	WorkAreaState^[WorkAreaNumber].Supporto := Forming^[1].Pallet;
	WorkAreaState^[WorkAreaNumber].F := 1;
	WorkAreaState^[WorkAreaNumber].ID 	:= ProgressiveNrWA^;
	ProgressiveNrWA^ := ProgressiveNrWA^ + 1;
	WorkAreaState^[WorkAreaNumber].P 	:= 0;
	WorkAreaState^[WorkAreaNumber].Slow := 1;
	WorkAreaState^[WorkAreaNumber].LGVAttr := Forming^[WorkAreaState^[WorkAreaNumber].F].LGVAttr;
	WorkAreaState^[WorkAreaNumber].State := WORKAREA_STATE_OCCUPIED_WORKING;
	
	InserisciNuovoPallet := FALSE;

ELSIF InserisciNuovoPallet AND WorkAreaState^[WorkAreaNumber].State < WORKAREA_STATE_OCCUPIED_WORKING AND FALSE THEN
	
	//Se la postazione ha codice fisso, lo assegno!
	IF CodicePostazione = 0 AND WorkAreaCodiciFissi[WorkAreaNumber] > 0 THEN
		CodicePostazione := WorkAreaCodiciFissi[WorkAreaNumber];
	END_IF

	(* Cerco Formatura *)
	IndiceFormaturaPostazione := 0;
	IndiceFormaturaPostazione := TFPalletizerGetFormingFromCodeSlab(Forming,CodicePostazione);
	//Assegno la formatura successivamanete nel WAManager
	IF IndiceFormaturaPostazione < 1 THEN
		IndiceFormaturaPostazione := 0;
		//Valuto la zona della postazione e ricavo la formatura in base alla zona di appartenenza	
	
		FOR cod:=1 TO MAXFORMINGCODE DO
			FormaturaZona[cod] := 0;
		END_FOR
		DoppiaFormaturaAttiva := FALSE;
		CodiceInFormaturaMem := 0;
		NumCodiciInFormaturaAttiviPerZona := 0;
		FOR zone:=1 TO MAXZONE DO
			FOR ar:=1 TO MAXAREA DO
				(* Verifico se la WorkArea appartiena ad una Zona *)
				IF WorkAreaZone.Zone[zone].WorkArea[ar] = WorkAreaNumber THEN
					FOR cod:=1 TO MAXFORMINGCODE DO
						IF FormaturaZona[cod] > 0 THEN
							DoppiaFormaturaAttiva := TRUE;
						END_IF
						FormaturaZona[cod] := TFPalletizerGetFormingFromCodeSlab(Forming,WorkAreaZone.Zone[zone].Code[cod]);
						IF WorkAreaZone.Zone[zone].Code[cod] <> CodiceInFormaturaMem  THEN//Memorizzo se ho un codice 
							NumCodiciInFormaturaAttiviPerZona := NumCodiciInFormaturaAttiviPerZona+1;
							CodiceInFormaturaMem := WorkAreaZone.Zone[zone].Code[cod];
						END_IF
					END_FOR
					EXIT;//Esco e vado a valutare le formature
				END_IF
			END_FOR
		END_FOR	
		FOR ar:=1 TO 4 DO
			FormaturePresenti[ar] := 0;
		END_FOR
		FOR ar:=1 TO MAXFORMINGCODE DO
		
			CASE FormaturaZona[ar] OF
				1:
					FormaturePresenti[1] := FormaturePresenti[1]+1; 	
				2:
					FormaturePresenti[2] := FormaturePresenti[2]+1;
				3:
					FormaturePresenti[3] := FormaturePresenti[3]+1;
				4:
					FormaturePresenti[4] := FormaturePresenti[4] +1;
			ELSE
				IndiceFormaturaPostazione := 0;			
			END_CASE				
		END_FOR
		//Cerco se nella zona ci sono + formature presenti, se è così codice formatura = 0, in modo che la macchina lo assagne in base alle esigenze
		//Altrimenti se solo una formatura è presente gli assegno quella!			
		IF FormaturePresenti[1] >= 1 THEN
			IF FormaturePresenti[2] >= 1 OR FormaturePresenti[3] >= 1 OR FormaturePresenti[4] >= 1 OR DoppiaFormaturaAttiva THEN
				IndiceFormaturaPostazione := 0;
			ELSE
				IndiceFormaturaPostazione := 1;
				IF NumCodiciInFormaturaAttiviPerZona = 1 THEN
					 CodicePostazione := CodiceInFormaturaMem;
				END_IF
			END_IF		
		ELSIF FormaturePresenti[2] >= 1 THEN
			IF FormaturePresenti[1] >= 1 OR FormaturePresenti[3] >= 1 OR FormaturePresenti[4] >= 1 OR DoppiaFormaturaAttiva THEN
				IndiceFormaturaPostazione := 0;
			ELSE
				IndiceFormaturaPostazione := 2;
				IF NumCodiciInFormaturaAttiviPerZona = 1 THEN
					 CodicePostazione := CodiceInFormaturaMem;
				END_IF
			END_IF		
		ELSIF FormaturePresenti[3] >= 1 THEN
			IF FormaturePresenti[2] >= 1 OR FormaturePresenti[1] >= 1 OR FormaturePresenti[4] >= 1 OR DoppiaFormaturaAttiva THEN
				IndiceFormaturaPostazione := 0;
			ELSE
				IndiceFormaturaPostazione := 3;
				IF NumCodiciInFormaturaAttiviPerZona = 1 THEN
					 CodicePostazione := CodiceInFormaturaMem;
				END_IF
			END_IF		
		ELSIF FormaturePresenti[4] >= 1 THEN
			IF FormaturePresenti[2] >= 1 OR FormaturePresenti[3] >= 1 OR FormaturePresenti[1] >= 1 OR DoppiaFormaturaAttiva THEN
				IndiceFormaturaPostazione := 0;
			ELSE
				IndiceFormaturaPostazione := 4;
				IF NumCodiciInFormaturaAttiviPerZona = 1 THEN
					 CodicePostazione := CodiceInFormaturaMem;
				END_IF
			END_IF		
		END_IF
	END_IF
	
	WorkAreaState^[WorkAreaNumber].Taped := -1;
	WorkAreaState^[WorkAreaNumber].LGV_ReqAbort := FALSE;
	IF AbilitaAssegnazioneCodicePiazzoleConPaccoSuRibaltino AND CodicePostazione = 0 THEN
		WorkAreaState^[WorkAreaNumber].Code := 0;
		WorkAreaState^[WorkAreaNumber].Initialize := TRUE;
	ELSE
		WorkAreaState^[WorkAreaNumber].Code := CodicePostazione;
		WorkAreaState^[WorkAreaNumber].Initialize := FALSE;
	END_IF
	WorkAreaState^[WorkAreaNumber].Supporto := Forming^[IndiceFormaturaPostazione].Pallet;
	WorkAreaState^[WorkAreaNumber].F := IndiceFormaturaPostazione;
	
	WorkAreaState^[WorkAreaNumber].ID := ProgressiveNrWA^;
	ProgressiveNrWA^ := ProgressiveNrWA^ + 1;
	WorkAreaState^[WorkAreaNumber].P := 0;
	WorkAreaState^[WorkAreaNumber].Slow := 1;
	WorkAreaState^[WorkAreaNumber].LGVAttr := Forming^[WorkAreaState^[WorkAreaNumber].F].LGVAttr;
	WorkAreaState^[WorkAreaNumber].State := WORKAREA_STATE_OCCUPIED_WORKING;

	InserisciNuovoPallet := FALSE;
END_IF

END_FUNCTION_BLOCK

// ---- POUs/TFPalletizerData/TFClearWorkAreaArray.TcPOU
FUNCTION TFClearWorkAreaArray : BOOL
VAR_INPUT
	WorkArea : POINTER TO ARRAY [1..MAXAREA] OF TFMachinePalletizer_WorkArea;
	WorkAreaState : POINTER TO ARRAY [1..MAXAREA] OF TFMachinePalletizer_WorkAreaState;
	k : uINT;
END_VAR
VAR
END_VAR

(* Copia dello stato delle WA in un backup *)
IF WorkAreaState^[k].ID > 0 THEN
	WorkAreaStateBK[k] := WorkAreaState^[k];
END_IF

WorkAreaState^[k] := EmptyWorkAreaState;
WorkAreaState^[k].State		:= WORKAREA_STATE_FREE_ENABLED;	(* Stato Area di Lavoro/Piazzola
																			(0=Assente e Area Disabilitata,
																			1=Presente e Area Disabilitata,
																			2=Assente in Lavorazione,
																			3=Presente in Lavorazione,
																			4=Presente con Pallettizzazione Terminata,
																			5=Presente con Pallettizzazione Terminata e Area Disabilitata,
																			6=Presente in Nastratura,
																			7=Presente in Nastratura e Area Disabilitata,
																			8=Presente con Nastratura Terminata,
																			9=Presente con Nastratura Terminata e Area Disabilitata,
																			10=Presente con Lavorazione Terminata,
																			11=Presente con Lavorazione Terminata e Area Disabilitata,
																			12=Presente con LGV in Richiesta Ingresso,
																			13=Presente con LGV in Richiesta Ingresso e Area Disabilitata,
																			14=Presente con LGV in Ingombro,
																			15=Presente con LGV in Ingombro e Area Disabilitata,
																			16=Presente con LGV Fuori Ingombro e Pallet Estratto,
																			17=Presente con LGV Fuori Ingombro e Pallet Estratto e Area Disabilitata, NOT USED !!!!!!!!!!!
																			99=Errore
																			-1 dato non valido) *)
																			
//TFClearWorkAreaStateSlab(WorkAreaState,k);																			
																			
WorkAreaState^[k].F					:= -1;	(* Forming Pointer - Puntatore tabella formature (1..n=, -1 dato non valido *)
WorkAreaState^[k].P					:= -1;	(* Pack Pointer - Puntatore tabella ELEMENTO (0..n-1=, -1 dato non valido),Numero ELEMENTO successivo da depositare *)
              
WorkAreaState^[k].Code				:= -1;	(* Codice di Pallettizzazione (0..n=, -1 dato non valido) x lastre, se Magazzino Falde, codice della falda *)
              
WorkAreaState^[k].PackPointerModified	:= FALSE;		(* Se TRUE, indica che è stata effettuata una modfica sui dati della WA da parte dell' HMI (Settata da HMI e resettata da PLC) *)
WorkAreaState^[k].PackPointer			:= -1;			(* Rappresenta l'indice del pacco da depositare dopo modfica manuale,cioè con PackPointerModified=TRUE *)

WorkAreaState^[k].Slab := EmptySlabArray;

WorkAreaState^[k].LGVAttr				:= 0;

TFClearWorkAreaBCRead(WorkAreaState);//Resetto i vari stati dl BARCODE

WorkAreaState^[k].H					:= 0.0; (* (mm) Altezza Reale. Viene calcolata dal PLC dopo ogni prelievo (Vuoti o Falde) o deposito Pallet e durante la pallettizzazione *)
WorkAreaState^[k].HPL				:= 0.0; (* (mm) Altezza del pallett utilizzato + altezza layers utilizzati *)

TFClearApprendimento(ADR(WorkAreaState^[k].Apprendimento));//Azzeramento apprendimento

(*
(* Apprendimenti nelle varie direzioni *)
WorkAreaState^[k].DoLearn_Y0		:= APPRENDIMENTO_DA_ESEGUIRE;	(* Stato apprendimento Direzione Y LATO 0° 0=Disabilitato, 1=Abilitato da Eseguire, 2=Eseguito, -1 dato non valido *)
WorkAreaState^[k].Learn_Y0			:= 0.0;	(* (mm) Quota inizio Apprendimento Direzione Y LATO 0° *)
WorkAreaState^[k].Learned_Y0		:= 0.0; (* Quota rilevata durante apprendimento Direzione Y LATO 0° *)

WorkAreaState^[k].DoLearn_Y180		:= APPRENDIMENTO_DA_ESEGUIRE;	(* Stato apprendimento Direzione Y LATO 180° 0=Disabilitato, 1=Abilitato da Eseguire, 2=Eseguito, -1 dato non valido *)
WorkAreaState^[k].Learn_Y180		:= 0.0;	(* (mm) Quota inizio Apprendimento Direzione Y LATO 180° *)
WorkAreaState^[k].Learned_Y180		:= 0.0; (* Quota rilevata durante apprendimento Direzione Y LATO 180° *)

WorkAreaState^[k].DoLearn_Z			:= APPRENDIMENTO_DA_ESEGUIRE;	(* Stato apprendimento Direzione Z 0=Disabilitato, 1=Abilitato da Eseguire, 2=Eseguito, -1 dato non valido *)
WorkAreaState^[k].Learn_Z			:= 0.0;	(* (mm) Quota inizio Apprendimento Direzione Z *)
WorkAreaState^[k].Learned_Z			:= 0.0; (* Quota rilevata durante apprendimento Direzione Z *)
*)
WorkAreaState^[k].RefuseLGV       	:= FALSE;	(* Abilitazione chiamata LGV a termine pallettizzazione - TRUE= Non chiama LGV quando pallet pieno, FALSE= viene eseguita richiesta LGV *)
              
WorkAreaState^[k].LGV_Req			:= 0;	(* Richiesta LGV (0=Nop, 1=Richiesta LGV, 2= Consenso Ingresso, -1= non valido) *)
WorkAreaState^[k].LGV_GetIn_GetOut	:= 0;	(* Tipo Richiesta LGV  (0=Nop, 1=Richiesta Prelievo, 2= Richiesta Deposito, -1= non valido) *)	
WorkAreaState^[k].LGV_ReqAbort		:= FALSE; (* Aborto chimata LGV *)


TFClearWorkAreaArray := TRUE;

END_FUNCTION

// ---- POUs/TFPalletizerData_Lastre/TFClearWorkAreaBCRead.TcPOU
FUNCTION TFClearWorkAreaBCRead : BOOL
VAR_INPUT
	WorkAreaState : POINTER TO TFMachinePalletizer_WorkAreaState;
END_VAR
VAR
	i : INT;
END_VAR

FOR i:=1 TO MAXNUMBARCODE DO
	WorkAreaState^.BCRead[i].State := LETTURA_ESEGUITA;
	WorkAreaState^.BCRead[i].Value := ''; 
	WorkAreaState^.BCRead[i].ErrorCode := 0;
END_FOR
TFClearWorkAreaBCRead := TRUE;

END_FUNCTION

// ---- POUs/TFPalletizerData_Lastre/TFClearApprendimento.TcPOU
FUNCTION TFClearApprendimento : BOOL //Funzione che pulisce la struttura dell'apprendimento
VAR_INPUT
	Apprendimento : POINTER TO TFMachinePalletizer_CoordinateApprendimento;
END_VAR
VAR
	i : INT;
END_VAR

MEMSET(ADR(Apprendimento^),0,SIZEOF(Apprendimento^));
TFClearApprendimento := TRUE;

END_FUNCTION

// ---- POUs/TFPalletizerData_Lastre/TFPalletizerGetFormingFromCodeSlab.TcPOU
FUNCTION TFPalletizerGetFormingFromCodeSlab : INT
VAR_INPUT
	Forming : POINTER TO ARRAY [1..MAXFORMING] OF TFMachinePalletizer_FormingForSlab;
	FCode : INT;
END_VAR
VAR
	pp : UINT;
	pf : INT;
	PCode : UINT;
END_VAR

(* Per Tutte le Formature Attive *)
FOR pf:=1 TO MAXFORMING DO
	IF Forming^[pf].Enable = 1 THEN
		(* Per tutti i codici di Pallettizzazione *)
		FOR pp:=1 TO MAXFORMINGCODE DO
			IF Forming^[pf].Code[pp] = FCode THEN
				TFPalletizerGetFormingFromCodeSlab := pf;
				RETURN;
			END_IF
		END_FOR
	END_IF
END_FOR
TFPalletizerGetFormingFromCodeSlab := 0;

END_FUNCTION

// ---- POUs/TFPalletizerDataTF/Utility Varie/TFCalcolaNumeroPostazioneDXSX.TcPOU
FUNCTION_BLOCK TFCalcolaNumeroPostazioneDXSX (* Restituisce il numero della postazione a DX e a SX rispetto alla poszione attuale della pinza *)
VAR_INPUT
	WorkArea 					: POINTER TO ARRAY[1..MAXAREA] OF TFMachinePalletizer_WorkArea; //Puntatore alla struttura WorkArea
	PosizioneAttuale			: LREAL;	//Posizione attuale dell'asse X
	DirezioneAsseX_Positiva		: BOOL;
END_VAR
VAR_OUTPUT
	NPostazioneDX : UINT;
	NPostazioneSX : UINT;
	PostazionePartenza : UINT;
END_VAR
VAR
	WADX: UINT;
	WASX: UINT;
	waDXSX : UINT;
END_VAR
(* Restituisce il numero della postazione a DX e a SX rispetto alla poszione attuale della pinza *)

WASX := 0;
WADX := 0;

CASE VERSO_PALLETTIZZATORE OF
	PALLETTIZZATORE_DX :
						FOR waDXSX := 1 TO MAXAREAPRESENT DO
							IF PosizioneAttuale > WorkArea^[waDXSX].X + 50  THEN
								WADX := WADX +1;
								IF WADX > MAXAREAPRESENT THEN
									WADX := MAXAREAPRESENT;
								END_IF
								NPostazioneDX		:= WADX;
								WorkAreaDX_Attuale  := WADX;
							ELSE
								WASX := WADX + 1;
								IF WADX = 0 THEN
									WADX:=1;
								END_IF
								IF WASX > MAXAREAPRESENT THEN
									WASX := MAXAREAPRESENT;
								END_IF
								NPostazioneSX		:= WASX;
								WorkAreaSX_Attuale := WASX;
								IF DirezioneAsseX_Positiva THEN
									PostazionePartenza:= WADX+1;
								ELSE
									PostazionePartenza:= WASX-1;
									
								END_IF
								EXIT;
							END_IF
						END_FOR					
						
	
	PALLETTIZZATORE_SX :
						CASE ORDINE_DISPOSIZIONE_POSTAZIONI OF

							CRESCENTE:
										FOR waDXSX := 1 TO MAXAREAPRESENT DO
											IF PosizioneAttuale > WorkArea^[waDXSX].X + 50  THEN
												WADX := WADX +1;
												IF WADX > MAXAREAPRESENT THEN
													WADX := MAXAREAPRESENT;
												END_IF
												NPostazioneDX		:= WADX;
												WorkAreaDX_Attuale  := WADX;
											ELSE
												WASX := WADX + 1;
												IF WADX = 0 THEN
													WADX:=1;
												END_IF
												IF WASX > MAXAREAPRESENT THEN
													WASX := MAXAREAPRESENT;
												END_IF
												NPostazioneSX		:= WASX;
												WorkAreaSX_Attuale := WASX;
												IF DirezioneAsseX_Positiva THEN
													
													//PostazionePartenza:= WADX;
													PostazionePartenza:= WASX;
												ELSE
													//PostazionePartenza:= WASX;
													PostazionePartenza:= WASX;
												END_IF
												EXIT;
											END_IF
										END_FOR
										
							DECRESCENTE:
										FOR waDXSX := MAXAREAPRESENT  TO 1 BY -1 DO
											IF PosizioneAttuale > WorkArea^[waDXSX].X THEN
												IF waDXSX = MAXAREAPRESENT THEN
													NPostazioneSX		:= 99;//Punto di prelievo
													WorkAreaSX_Attuale  := 99;
													NPostazioneDX		:= waDXSX;
													WorkAreaDX_Attuale  := waDXSX;
												ELSIF waDXSX = 1 THEN
													NPostazioneSX		:= 1;
													NPostazioneDX		:= 1;
													WorkAreaSX_Attuale  := 1;
													WorkAreaDX_Attuale  := 1;
													IF DirezioneAsseX_Positiva THEN
														PostazionePartenza:= WorkAreaDX_Attuale;
													ELSE
														PostazionePartenza:= WorkAreaSX_Attuale;
													END_IF
													EXIT;
												ELSE
													NPostazioneSX		:= waDXSX+1;
													NPostazioneDX		:= waDXSX-1;
													WorkAreaSX_Attuale  := waDXSX;
													WorkAreaDX_Attuale	:= waDXSX;
												END_IF	
												
											ELSIF PosizioneAttuale <= WorkArea^[waDXSX].X THEN
												IF waDXSX = MAXAREAPRESENT THEN
													NPostazioneSX		:= 99;//Punto di prelievo
													NPostazioneDX		:= waDXSX;
													WorkAreaSX_Attuale  := waDXSX;
													WorkAreaDX_Attuale  := waDXSX;
													IF DirezioneAsseX_Positiva THEN
														PostazionePartenza:= WorkAreaDX_Attuale;
													ELSE
														PostazionePartenza:= WorkAreaSX_Attuale;
													END_IF
													EXIT;
												ELSIF waDXSX = 1 THEN
													NPostazioneSX		:= waDXSX+1;
													NPostazioneDX		:= 1;
													WorkAreaSX_Attuale  := waDXSX;
													WorkAreaDX_Attuale  := waDXSX;
												ELSE
													NPostazioneSX		:= waDXSX+1;
													NPostazioneDX		:= waDXSX-1;
													WorkAreaSX_Attuale  := waDXSX;
													WorkAreaDX_Attuale	:= waDXSX;
													IF DirezioneAsseX_Positiva THEN
														PostazionePartenza:= WorkAreaDX_Attuale;
													ELSE
														PostazionePartenza:= WorkAreaSX_Attuale;
													END_IF
													EXIT;
												END_IF
												
											END_IF
										END_FOR	
										
						END_CASE
	
	
END_CASE

END_FUNCTION_BLOCK

// ---- Data types/AlbertoPruevas/Funciones/Fun_SensoresTasteggio.TcPOU
FUNCTION Fun_SensoresTasteggio : BOOL
VAR_INPUT
	Sensor_Tasteo_1 				: BOOL ;
	Sensor_Tasteo_2 				: BOOL ;
	Sensor_Tasteo_3 				: BOOL ;
	Sensor_Tasteo_4 				: BOOL ;
	Nu_sensores_Dar_Out				: BYTE ;
END_VAR
VAR_OUTPUT
	Sensores_Tasteggio_Ok 			: BOOL ;
	Nu_Sesores_Activos				: BYTE ;
END_VAR
VAR
END_VAR

Nu_Sesores_Activos := BOOL_TO_BYTE(Sensor_Tasteo_1) + BOOL_TO_BYTE(Sensor_Tasteo_2) + BOOL_TO_BYTE(Sensor_Tasteo_3) + BOOL_TO_BYTE(Sensor_Tasteo_4) ; 

IF Nu_Sesores_Activos >= Nu_sensores_Dar_Out THEN
	Sensores_Tasteggio_Ok := TRUE ;
	ELSE
	Sensores_Tasteggio_Ok := FALSE ;	
	
END_IF

END_FUNCTION

// ---- Data types/AlbertoPruevas/Funciones/Fun_PiezaLadoCaballete.TcPOU
FUNCTION Fun_PiezaLadoCaballete : Uint
VAR_INPUT
	Nu_PiezaGlobal 			: UINT ;
	Grados 					: pointer TO UINT ;
END_VAR
VAR_OUTPUT
	Nu_pieza_LadoA: UINT;
	Nu_pieza_LadoB: UINT;
END_VAR
VAR
	
	RestoDiv: UINT;
END_VAR



//Dia 23-10-2025
CASE Nu_PiezaGlobal OF
	1:
		Nu_pieza_LadoA :=  Nu_PiezaGlobal ;
		Grados^ := 0;
	2..100 :
		IF Nu_PiezaGlobal > 1 THEN 
			RestoDiv := Nu_PiezaGlobal MOD 2 ;
			CASE RestoDiv OF
				0:
					Nu_pieza_LadoB := Nu_PiezaGlobal / 2 ;
					Grados^ := 180;
				1:
					Nu_pieza_LadoA := ((Nu_PiezaGlobal-1) / 2)+1 ;
					Grados^ := 0;	
			END_CASE
		END_IF
END_CASE

END_FUNCTION

// ---- POUs/TFLGV/GateAccessLGV.TcPOU
FUNCTION_BLOCK GateAccessLGV
VAR_INPUT
	WorkArea 				: POINTER TO ARRAY [1..MAXAREA] OF TFMachinePalletizer_WorkArea;
	WorkAreaState 			: POINTER TO ARRAY [1..MAXAREA] OF TFMachinePalletizer_WorkAreaState;//WorkAreaState 			: POINTER TO TFMachinePalletizer_WorkAreaState;
	PH_WorkArea 			: BOOL;//FTC Presenza elemento
	LGV_InfeedReq_HW 		: BOOL;//Richiesta ingresso cablata
	LGV_Encumbrance_HW 		: BOOL;//Ingombro cablato
	LGV_InfeedReq_SW 		: BOOL;//Richiesta ingresso SW
	LGV_Encumbrance_SW 		: BOOL;//Ingombro SW
	LGV_HW_SW_SWITCH 		: BOOL := FALSE;//tipologia di scambio consensi true= cablata, false= software
	Machine					: POINTER TO TFMachinePalletizer_TF; //Macchina
	TimeBase 				: REAL;//Tempo base PLC
	OtherAccessActive 		: BOOL;//Altri gate access attivi
	Modules	 				: POINTER TO TFPalletizerModules;
	OtherMachineStopPresent	: BOOL; //presenza altra macchina per considerare il suo stop in fase
	OtherMachineStopDone 	: BOOL;//stop eseguito di altre macchine collegate 	
	LGV_Data 				: POINTER TO ARRAY [1..MAXAREA] OF ST_SupervisorData;//Puntatore alla struttura dati relativi alla chiamata della postazione
	IndicePostazione		: UINT;
END_VAR
VAR_OUTPUT
	Logic_Req 			: BOOL;	(* Bit di richiesta logia da parte della postazione *)
	LGV_InfeedRequest 	: BOOL; (* Bit di segnalazione di richiesta ingresso da veicolo *)
	LGV_InfeedOk 		: BOOL; (* Segnalazione accesso consentito *)
	LGVAccessLamp 		: BOOL; (* Access Lamp: 	OFF = No Access Consent,
										ON = Access Consent,
										FLASH (1sec) = Access Requested (Machine Stopping)
										FLASH (0.5sec) = Waiting Restart
										FLASH (0.1sec) = Access Error *)
										
	LGVAccesActive 		: BOOL; (* Gate Acces Sequence in Execution *)
	OtherMachineStopReq : BOOL;	
	
	LGVResetHSKSUPNAV 	: BOOL;	
	LGV_ResetSW_RicIng 	: BOOL;
	
	ErrAck 			: BOOL; //Error Acknowledge Safaty
	ErrAckDriver 	: BOOL; //Error Acknowledge Drive
	ErrorCode 		: UINT; //Codice di errore
	ReqPowerOffSimulation : bool;//Richiesta di power OFF x simulazione senza HW
END_VAR
VAR
	LGVCase : INT;
	j : UINT;
	k : UINT; 
	LGV_REQIN : BOOL;// bit di richiesta utilizzato all'interno del FB
	LGV_Encumbrance : BOOL;//Bit di ingombro utilizzato all'interno del FB
	Power 				: BOOL;
	
	
	ParametersArray : ParametersArray;
	//LGVAccessOK : BOOL;
	LGVAccessERROR : BOOL;	
	LGVAccessReqIN : BOOL;
	MachineWasRunning : BOOL;
	Timer100 : REAL;
	Timer200 : REAL;
	Timer1000 : REAL;
	Clock100 : BOOL;
	Clock200 : BOOL;
	Clock1000 : BOOL;
	TimerMachineWaitRunning : REAL;
	TimerPowerOFF : REAL;
	TimeoutControlloBarriereSicurezza : REAL;
	TimerOkBarriereSicurezze : REAL;
	TimeoutAnomaliaConsensi : REAL;
	TimerRitardoPower:REAL;
	AggiornaDatiPostazione : BOOL;//se true, quando va via la richiesta e l'ingombro aggiorniamo i dati
END_VAR

TFTimerCall(ADR(Timer100),TimeBase);
TFTimerCall(ADR(Timer200),TimeBase);
TFTimerCall(ADR(Timer1000),TimeBase);
TFTimerCall(ADR(TimerMachineWaitRunning),TimeBase);
TFTimerCall(ADR(TimerPowerOFF),TimeBase);
TFTimerCall(ADR(TimeoutControlloBarriereSicurezza),TimeBase);
TFTimerCall(ADR(TimerOkBarriereSicurezze),TimeBase);
TFTimerCall(ADR(TimeoutAnomaliaConsensi),TimeBase);
TFTimerCall(ADR(TimerRitardoPower),TimeBase);

(* A seconda della tipologia dei consensi, valorizzo le variabili interne*)
IF NOT LGV_HW_SW_SWITCH THEN
	LGV_REQIN 		:= LGV_InfeedReq_HW;
	LGV_Encumbrance := LGV_Encumbrance_HW;
ELSE	
	LGV_REQIN 		:= LGV_InfeedReq_SW;
	LGV_Encumbrance := LGV_Encumbrance_SW;
END_IF

(* Setto il bit interno di Power *)
Power := Machine^.IN.PowerOk;
(* Setto il valore dello stop in fase della macchina esterna se non è presente *)
IF NOT OtherMachineStopPresent THEN
	OtherMachineStopDone := OtherMachineStopReq;
END_IF

IF IndicePostazione <= 0 THEN
	RETURN;
END_IF

CASE LGVCase OF

	(* Case 0 *)
	0:	
		ReqPowerOffSimulation       := FALSE;
		ErrorCode 					:= 0;
		LGVResetHSKSUPNAV 			:= FALSE;
		LGVAccesActive 				:= FALSE;
		LGV_InfeedOk 				:= FALSE;
		LGVAccessReqIN 				:= FALSE;
		OtherMachineStopReq 		:= FALSE;
		Logic_Req 					:= FALSE;
		IF (WorkAreaState^[IndicePostazione].State = WORKAREA_STATE_OCCUPIED_LGVREQ OR WorkAreaState^[IndicePostazione].State = WORKAREA_STATE_FREE_LGVREQ) AND 
			WorkArea^[IndicePostazione].Enable = 1 AND WorkAreaState^[IndicePostazione].LGV_Req = 1 AND NOT LGV_Data^[IndicePostazione].HskToSupervisor.DisableLGV THEN
				Logic_Req 				:= TRUE;
		END_IF		
		// Command Case = 15 is WorkFlowsRunning after Homing WorkFlow NOTES: State=DO_RUN+1 it will be better!!!!
		MachineWasRunning := Machine^.CmdExe.Code = CmdDO AND Machine^.CmdExe.CmdCase = 15 AND Machine^.CmdExe.PhaseStopRequest = 0 AND Machine^.CmdExe.RapidStopRequest = 0;
		TFTimerSet(ADR(TimerMachineWaitRunning),1000,NOT MachineWasRunning);
		
		IF LGV_REQIN AND Logic_Req AND NOT OtherAccessActive AND MachineWasRunning AND TFTimerDone(ADR(TimerMachineWaitRunning)) THEN
			LGVAccesActive 	:= TRUE;
			LGVAccessERROR 	:= FALSE;
			LGVAccessReqIN 	:= TRUE;
			(* Machine Was Running if CmdDO and No Stop Request *)
			LGVCase 		:= LGVCase + 1;
			AggiornaDatiPostazione := TRUE;
		END_IF	
			
	(* Case 1 - Phase Stop *)
	1:	TFParametersArrayClear(ADR(ParametersArray));
		TFCommandSend(CmdSTOPPHASE,ParametersArray,Machine^.Cmd);
		OtherMachineStopReq 		:= TRUE;
		AggiornaDatiPostazione 		:= TRUE;
		LGVCase 					:= LGVCase + 1;
		
	(* Case 2 - Cmd DO END *)	
	2:	IF ((TFStateCodeGet(Machine^.State) = StateDO_END AND NOT
			TFIsModuleError(Machine^.Error)) OR
			Machine^.CmdExe.Code = CmdNOP)  THEN
			TFTimerSet(ADR(TimerPowerOFF),1000,TRUE);
			LGVCase := LGVCase + 1;
		ELSIF TFIsModuleError(Machine^.Error) OR 
			TFPalletizerIsModuleError(Modules) THEN
			LGVCase := 0; 
		END_IF

	(* Case 3 - Power Off *)
	3:	IF TFTimerDone(ADR(TimerPowerOFF)) AND OtherMachineStopDone THEN
			TFParametersArrayClear(ADR(ParametersArray));
			ParametersArray.Parameters[0] := '0';
			TFCommandSend(CmdPOWER,ParametersArray,Machine^.Cmd);
			LGVCase := LGVCase + 1;
		END_IF	

	(* Case 4 - Power Off OK *)	
	4:	ReqPowerOffSimulation := TRUE;
		IF (TFStateCodeGet(Machine^.State) = StatePOWER_END) AND// OR NOT Power) AND
			NOT TFIsModuleError(Machine^.Error) AND 
			NOT TFPalletizerIsModuleError(Modules) AND 
			NOT OtherAccessActive THEN
			LGVCase := LGVCase + 1;
		ELSIF NOT LGV_REQIN THEN
			LGVCase := 6;
		ELSIF TFIsModuleError(Machine^.Error) THEN
			LGVCase := 0;
		END_IF
		TFTimerSet(ADR(TimeoutAnomaliaConsensi),120000,TRUE);
		
	(* Case 5  LGV IN *)
	5:	
		
		IF LGV_REQIN AND Logic_Req AND NOT TFIsModuleError(Machine^.Error)THEN
			LGV_InfeedRequest := TRUE;
			LGVAccessReqIN := FALSE;
			LGV_InfeedOk := TRUE;
			TFTimerSet(ADR(TimeoutAnomaliaConsensi),300000,TRUE);
		ELSE
			LGV_InfeedRequest := FALSE;
			LGV_InfeedOk := FALSE;
			LGVAccessReqIN := FALSE;
		END_IF
		
		IF NOT LGV_REQIN AND NOT LGV_Encumbrance THEN
			LGV_InfeedRequest := FALSE;
			LGVCase := LGVCase + 1;
		ELSIF TFTimerDone(ADR(TimeoutAnomaliaConsensi)) AND ((LGV_REQIN AND NOT LGV_Encumbrance) OR (NOT LGV_REQIN AND LGV_Encumbrance)) THEN
			LGV_InfeedReq_SW := FALSE;
			LGV_Encumbrance_SW := FALSE;
			LGV_REQIN := LGV_InfeedReq_SW;
			LGV_Encumbrance := LGV_Encumbrance_SW;
			LGVResetHSKSUPNAV := TRUE;
			ErrorCode := ErrMACHINEPALLETIZER_ANOMALIA_CONSENSI_SUPNAVETTE;
			LGVCase := 0;
		END_IF
		IF TFIsModuleError(Machine^.Error) THEN // se la macchina è in errore, forzo l'uscita da questo stato
			LGV_InfeedReq_SW 	:= FALSE;
			LGV_Encumbrance_SW 	:= FALSE;
			LGV_REQIN 			:= LGV_InfeedReq_SW;
			LGV_Encumbrance 	:= LGV_Encumbrance_SW;
			LGVResetHSKSUPNAV 	:= TRUE;
			ErrorCode := ErrMACHINEPALLETIZER_AZZERAMENTO_FORZATO_RICHIN_SUPNAVETTE;
			LGVCase := 0;
		END_IF	
		TFTimerSet(ADR(TimeoutControlloBarriereSicurezza),20000,TRUE);

	(* Case 6 - *)
	6:	
		IF TFIsModuleError(Machine^.Error) THEN // se la macchina è in errore, forzo l'uscita da questo stato
			LGV_InfeedReq_SW := FALSE;
			LGV_Encumbrance_SW := FALSE;
			LGV_REQIN := LGV_InfeedReq_SW;
			LGV_Encumbrance := LGV_Encumbrance_SW;
			LGVResetHSKSUPNAV := TRUE;
			ErrorCode := ErrMACHINEPALLETIZER_AZZERAMENTO_FORZATO_RICHIN_SUPNAVETTE;
			LGVCase := 0;
		ELSE
			LGVCase := 10;	
		END_IF
		
	(* Case 7 - Power ON *)
	10:	IF NOT OtherAccessActive AND TFTimerDone(ADR(TimerOkBarriereSicurezze))  THEN
			TFTimerSet(ADR(TimerRitardoPower),100,TRUE);
			LGVCase := LGVCase + 1;	
		ELSIF OtherAccessActive THEN
			LGVCase := 0;
		ELSIF TFTimerDone(ADR(TimeoutControlloBarriereSicurezza)) THEN
			ErrorCode := ErrMACHINEPALLETIZER_BARRIEREOCCUPATE_LGVREQ_OFF;
			LGVCase := 0;
		END_IF
		IF TFIsModuleError(Machine^.Error) THEN // se la macchina è in errore, forzo l'uscita da questo stato
			LGV_InfeedReq_SW := FALSE;
			LGV_Encumbrance_SW := FALSE;
			LGV_REQIN := LGV_InfeedReq_SW;
			LGV_Encumbrance := LGV_Encumbrance_SW;
			LGVResetHSKSUPNAV := TRUE;
			ErrorCode := ErrMACHINEPALLETIZER_AZZERAMENTO_FORZATO_RICHIN_SUPNAVETTE;
			LGVCase := 0;
		END_IF
(**************************************************************************)
(**************** Error Acknowledge Safety + AZIONAMENTI ***************************)
	11:
		IF TFTimerDone(ADR(TimerRitardoPower)) THEN
			TFTimerSet(ADR(TimerRitardoPower),100,TRUE);
			ErrAck := TRUE;
			LGVCase := LGVCase + 1;	
		END_IF
	
	12:	
		IF TFTimerDone(ADR(TimerRitardoPower)) THEN
			TFTimerSet(ADR(TimerRitardoPower),100,TRUE);
			ErrAck := FALSE;
			LGVCase := LGVCase + 1;	
		END_IF

	13:
		IF TFTimerDone(ADR(TimerRitardoPower)) THEN
			TFTimerSet(ADR(TimerRitardoPower),100,TRUE);
			ErrAckDriver := TRUE;
			LGVCase := LGVCase+1;
		END_IF
		
	14:
		IF TFTimerDone(ADR(TimerRitardoPower)) THEN
			TFTimerSet(ADR(TimerRitardoPower),100,TRUE);
			ErrAckDriver := FALSE;
			LGVCase := LGVCase+1;
		END_IF

	15: 
		IF TFTimerDone(ADR(TimerRitardoPower)) THEN
			LGVCase := 20;
		END_IF
(**************************************************************************)
(**************************************************************************)		
	(* Case 20 - Power ON *)
	20:	IF NOT OtherAccessActive AND TFTimerDone(ADR(TimerOkBarriereSicurezze)) THEN
			TFParametersArrayClear(ADR(ParametersArray));
			ParametersArray.Parameters[0] := '1';
			TFCommandSend(CmdPOWER,ParametersArray,Machine^.Cmd);
			LGV_ResetSW_RicIng := TRUE;
			LGVCase := LGVCase + 1;	
		ELSIF TFTimerDone(ADR(TimeoutControlloBarriereSicurezza)) THEN
			ErrorCode := ErrMACHINEPALLETIZER_BARRIEREOCCUPATE_LGVREQ_OFF;
			LGVCase := 0;
		END_IF	
		IF TFIsModuleError(Machine^.Error) THEN // se la macchina è in errore, forzo l'uscita da questo stato
			LGV_InfeedReq_SW := FALSE;
			LGV_Encumbrance_SW := FALSE;
			LGV_REQIN := LGV_InfeedReq_SW;
			LGV_Encumbrance := LGV_Encumbrance_SW;
			LGVResetHSKSUPNAV := TRUE;
			ErrorCode := ErrMACHINEPALLETIZER_AZZERAMENTO_FORZATO_RICHIN_SUPNAVETTE;
			LGVCase := 0;
		END_IF
			
	(* Case 21 - Power On OK *)
	21:	
		ReqPowerOffSimulation := FALSE;
		IF TFStateCodeGet(Machine^.State) = StatePOWER_END OR
			TFIsModuleError(Machine^.Error) THEN
			LGV_ResetSW_RicIng := FALSE;
			LGVCase := LGVCase + 1;	
		END_IF
		
	(* Case 22 - Cmd DO *)
	22:	
		IF MachineWasRunning AND
			Machine^.IN.Mode.Auto AND
			NOT Machine^.IN.Mode.StopRequest AND
			NOT Machine^.IN.Mode.RapidStopRequest AND NOT OtherAccessActive THEN
			(*AND (SecurityGateStatus OR NOT ControlGateSecurity^*) 
			TFParametersArrayClear(ADR(ParametersArray));
			TFCommandSend(CmdDO,ParametersArray,Machine^.Cmd);
			OtherMachineStopReq := FALSE;
		END_IF
		LGVCase := 0;
	
	ELSE
		LGVAccessERROR := TRUE;
		LGVCase := 0;
	
END_CASE

(* In base allo stato dell'ingombro del veicolo e delle ftc vado a valorizzare/sbiancare i valori *)
IF NOT LGV_REQIN AND NOT LGV_Encumbrance AND AggiornaDatiPostazione THEN
	AggiornaDatiPostazione := FALSE;//Abbasso la richiesta di aggiornamento dati postazione
	CASE WorkAreaState^[IndicePostazione].LGV_GetIn_GetOut OF
		REQ_PRELIEVO_LGV_PIENO:
								IF NOT PH_WorkArea THEN
									// Pulisco piazzola in seguito ad estrazione
									TFClearWorkAreaArray(WorkArea,WorkAreaState,IndicePostazione);
									I_PHPresenzaPalletVirtuale[IndicePostazione]:=FALSE;
								ELSE
									;
								END_IF	
		REQ_PRELIEVO_LGV_VUOTO:
								IF NOT PH_WorkArea THEN
									// Pulisco piazzola in seguito ad estrazione
									TFClearWorkAreaArray(WorkArea,WorkAreaState,IndicePostazione);
									I_PHPresenzaPalletVirtuale[IndicePostazione]:=FALSE;
								ELSE
									;
								END_IF
			
		REQ_DEPOSITO_LGV_VUOTO:
								IF NOT PH_WorkArea AND NOT SIMULAZIONE_NO_HW THEN
									// Pulisco piazzola in seguito ad estrazione
									TFClearWorkAreaArray(WorkArea,WorkAreaState,IndicePostazione);
									I_PHPresenzaPalletVirtuale[IndicePostazione]:=FALSE;
								ELSE
									CASE WorkArea^[IndicePostazione].Typology OF
		
										TYPOLOGY_PALLET:
														WorkAreaState^[IndicePostazione].Supporto.Code 	:= LGV_Data^[IndicePostazione].DataElementFromSupervisor.SupportType;
										
										TYPOLOGY_WASTE:
														WorkAreaState^[IndicePostazione].Supporto.Code 		:= CodeWasteSupport;//LGV_Data^.DataElementFromSupervisor.SupportType;
														WorkAreaState^[IndicePostazione].Supporto.Tipologia  	:= TYPOLOGY_WASTE;
														WorkAreaState^[IndicePostazione].Supporto.Code		:= CodeWasteSupport;	//Codice del pallet	
														WorkAreaState^[IndicePostazione].Code					:= 3;
																																			 
										TYPOLOGY_LAYER:
														WorkAreaState^[IndicePostazione].Supporto.Code 	:= LGV_Data^[IndicePostazione].DataElementFromSupervisor.LayerData.Code;
														WorkAreaState^[IndicePostazione].LayerData		:= LGV_Data^[IndicePostazione].DataElementFromSupervisor.LayerData;
										
									END_CASE
									ProgressiveNrWA 	:= ProgressiveNrWA+1;
									WorkAreaState^[IndicePostazione].ID 	:= ProgressiveNrWA; 
								END_IF
								
			
		REQ_DEPOSITO_LGV_PIENO:
								IF NOT PH_WorkArea AND NOT SIMULAZIONE_NO_HW THEN
									// Pulisco piazzola in seguito ad estrazione
									TFClearWorkAreaArray(WorkArea,WorkAreaState,IndicePostazione);
									I_PHPresenzaPalletVirtuale[IndicePostazione]:=FALSE;
								ELSE
									CASE WorkArea^[IndicePostazione].Typology OF
	
										TYPOLOGY_PALLET:
														WorkAreaState^[IndicePostazione].Supporto.Code 	:= LGV_Data^[IndicePostazione].DataElementFromSupervisor.SupportType;
										
										TYPOLOGY_WASTE:
														WorkAreaState^[IndicePostazione].Supporto.Code 		:= CodeWasteSupport;//LGV_Data^.DataElementFromSupervisor.SupportType;
														WorkAreaState^[IndicePostazione].Supporto.Tipologia  	:= TYPOLOGY_WASTE;
														WorkAreaState^[IndicePostazione].Supporto.Code		:= CodeWasteSupport;	//Codice del pallet	
														WorkAreaState^[IndicePostazione].Code					:= CodeWasteSupport;
																																			 
										TYPOLOGY_LAYER:
														WorkAreaState^[IndicePostazione].Supporto.Code 	:= LGV_Data^[IndicePostazione].DataElementFromSupervisor.LayerData.Code;
														WorkAreaState^[IndicePostazione].LayerData		:= Actual_WorkOrder.Layer;//  LGV_Data^[IndicePostazione].DataElementFromSupervisor.LayerData;
										
									END_CASE
									ProgressiveNrWA 	:= ProgressiveNrWA+1;
									WorkAreaState^[IndicePostazione].ID 	:= ProgressiveNrWA; 
								END_IF
	END_CASE
END_IF

(* Clocks *)
IF TFTimerDone(ADR(Timer100)) THEN
	TFTimerSet(ADR(Timer100),100,TRUE);
	Clock100 := NOT Clock100;
END_IF
IF TFTimerDone(ADR(Timer200)) THEN
	TFTimerSet(ADR(Timer200),200,TRUE);
	Clock200 := NOT Clock200;
END_IF
IF TFTimerDone(ADR(Timer1000)) THEN
	TFTimerSet(ADR(Timer1000),1000,TRUE);
	Clock1000 := NOT Clock1000;
END_IF

(* Access Lamp *)
LGVAccessLamp := ((LGV_InfeedOk AND Clock200) OR
				//(AccessReqOUT AND Clock500) OR
				(LGVAccessReqIN AND Clock1000))AND
				NOT LGVAccessERROR OR (LGVAccessERROR AND Clock100);

END_FUNCTION_BLOCK

// ---- POUs/TFMachines/TFMachinePalletizer_TF.TcPOU
FUNCTION_BLOCK TFMachinePalletizer_TF
VAR_INPUT
	Cmd 		: CommandBuffer;
	Cfg 		: Config;
	IN  		: TFMachinePalletizer_IN;
	
	Modules 					: POINTER TO TFPalletizerModules;
	
	WorkSpace 					: POINTER TO TFMachinePalletizer_WorkSpace;
	WorkFootprint 				: POINTER TO ARRAY [1..MAXFOOTPRINT] OF TFMachinePalletizer_WorkFootprint;
	WorkPickPoint 				: POINTER TO ARRAY [1..MAXPICKPOINT] OF TFMachinePalletizer_WorkPickPointSlab;
	WorkPickPointState 			: POINTER TO ARRAY [1..MAXPICKPOINT] OF TFMachinePalletizer_WorkPickPoint_State;
	//WorkPickPointTransportState	: POINTER TO ARRAY [1..MAXPICKPOINT] OF TFMachinePalletizer_WorkPickPointTransport_State;
	//WorkPickPointStoreState		: POINTER TO ARRAY [1..MAXPICKPOINT] OF TFMachinePalletizer_WorkPickPointStore_State;
	WorkPickPointDimension 		: POINTER TO ARRAY [1..MAXPICKPOINT] OF Work_PickPoint_Dimension;
	WorkPickPointOffset 		: POINTER TO ARRAY [1..MAXPICKPOINT] OF TFMachinePalletizer_WorkPickPointOffset;
	
	WorkArea 					: POINTER TO ARRAY [1..MAXAREA] OF TFMachinePalletizer_WorkArea;
	WorkAreaState 				: POINTER TO ARRAY [1..MAXAREA] OF TFMachinePalletizer_WorkAreaState;
	WorkAreaOffset 				: POINTER TO ARRAY [1..MAXAREA] OF TFMachinePalletizer_WorkAreaOffset;
	WAPointer 					: ARRAY [1..MAXAREA] OF TFMachinePalletizer_WorkAreaSort;			
	AxisOverride 				: POINTER TO TFMachinePalletizer_VelocityOverride_TF;			//Indica la struttura degli Override
	Pallet 						: POINTER TO ARRAY [1..MAXPALLET] OF TFMachinePalletizer_Pallet;		//Indica la struttura dei Pallet
	Layer 						: POINTER TO ARRAY [1..MAXLAYER] OF TFMachinePalletizer_Layer;		//Indica la struttura delle falde
	Forming 					: POINTER TO ARRAY [1..MAXFORMING] OF TFMachinePalletizer_FormingForSlab; //Indica la Struttura delle formature
	//AxisParK 					: POINTER TO Ax_Palletizer_Parameters;	//Parametri asse K
	
	ManCmd 						: POINTER TO TFModulePalletizerRobot_ManCmd;
	Mission 					: POINTER TO TFMachinePalletizer_Mission;	//Indica la missione in esecuzione
	Traiettoria 				: POINTER TO TFTraiettoria;				//Indica i parametri della traiettoria
	
	PickPlaceParameters			: POINTER TO TFMachinePalletizer_PickPlaceParameters;// Parametri Presa&Rilascio Piastrella/Falda/Pallet
	MachineManCmd 				: POINTER TO TFMachinePalletizer_ManCmd;
	ProgressiveNrWA 			: POINTER TO UDINT;
	UsedCode 					: POINTER TO ARRAY [1..MAXFORMINGCODE] OF INT;
	TCPParameter 				: POINTER TO TFModulePalletizerRobot_TCPPar;				// Indica i parametri delle manine(solitamente è valorizzata l'altezza "Z")
	TilterPack 					: POINTER TO ARRAY [1..MAXHANDLINGSTACK] OF TFHandlingPack;	// Indica il pacco presente sul ribaltino
	//UniqueCycle : BOOL;
	PreviousPWA 				: POINTER TO INT;
	RestoreCWA 					: POINTER TO BOOL;
	//TouchErrorEnable : BOOL;
	GateAccesExecuted 			: BOOL;
	PreviousStackWA 			: POINTER TO INT;
	WorkAreaZone 				: POINTER TO TFMachinePalletizer_WorkAreaZone; // Indica la suddivisione a zone delle WorkArea
	//HandlingPackTable : POINTER TO TFHandlingPackTable; 		// Tabella dei pacchi presenti sui trasporti
	ArrayPacchi 				: POINTER TO DUT_ArrayPacchi; 					//Array contenente i pacchi sui trasporti				

	PX_GripPresence 			: BOOL; //Fotocellula presenza Materiale su pinza
	
	WorkAreaManager 			: POINTER TO TFWorkAreaManager;	// Gestore delle Missioni e delle WorkArea
	MissionStateCase 			: POINTER TO MissionStateCase;	// Stato Delle Missioni 
	AbilitaControlloPHGripPresence 	: BOOL; 	// Se TRUE = Abilita il controllo della fotocellula di presenza materiale sulla pinza
	//AbilitaControlloCoppia 			: BOOL;			// Se TRUE = Disabilita il controllo della coppia
	AbilitaAnticipoDinamico 		: POINTER TO BOOL;				// Se TRUE = Abilitazione dell'anticipo dinamico dei movimienti
	AbilitaCalcoloIngombroOttimizzato   : POINTER TO BOOL;				// Se TRUE = Abilitazione del calcolo degli ingombri utilizzando l'angolo di rotazione attuale della pinza
	GestioneAZoneAbilitata 				: POINTER TO BOOL; //Abilitazione della gestione zone
	AbilitaDepositoPaccoOrrizzonataleConTasteggio : POINTER TO BOOL;
	AbilitaInterpolazioneAssi 	: POINTER TO BOOL; 			// Se TRUE = Abilitazione dell'interpolazione degli assi
	STARTInterpolazioneASSI 	: POINTER TO BOOL;			// Se TRUE = Lancia l'interpolazione degli assi
	AbilitaDisposizionePalletContinua : POINTER TO BOOL; 	// Se TRUE = abilita il deposito dei pallet in modo continuo
	AbilitaForzaturaStatoWAMDaCicloRiposoACicloPrelievo : POINTER TO BOOL; // Se TRUE = forza lo stato del WAM da cilco di riposo a ciclo di prelievo pacco
	AbilitaOffsetInUscitaTasteggioPrelievoPallet : POINTER TO BOOL; // Abilitazione dell'offset in uscita dei tastatori in prelievo pallet con tasteggio
	AbilitaAccostamentoAsseZ : POINTER TO BOOL; // Abilitazione dell'accostamento ell'asse Z.. Se TRUE : Ad una certa quota l'asse si muove in lenta
	AbilitaErroreComunicazioneTrasporti : BOOL; //Abilitazione Errore di comunicazione con i trasporti
	SimulazioneSenzaPalletFalde : BOOL;
	//MaterialeDepositatoSuLinea : POINTER TO BOOL;
	WorkAreaProductionList : POINTER TO ARRAY [1..MAXAREA] OF TFMachinePalletizer_ListaProduzione_WAM;
	RichiestaIngZonaDX : BOOL;
	RichiestaIngZonaSX : BOOL;
END_VAR
VAR_OUTPUT
	CmdExe : CommandExe;
	CmdExd : CommandExe;
	CmdNext : Command;
	CmdLog : CommandLog;
	State : State;
	StateLog : StateLog;
	Error : Error;
	ErrorLog : ErrorLog;
	Warning : Warning;
	WarningLog : WarningLog;
	OUT : TFMachinePalletizer_OUT;
	PalletStackEmpty : INT;
	LayerStackEmpty : INT;
	AllWABusy : INT;
	AssiInterpolati 			: BOOL;
	PinzaInQuotaFuoriIngombroPerTrasporti : BOOL;// la Quota della pinza mi garantisce che sono in fuori ingombro e il ribaltino può ruotare
END_VAR
VAR
	Init : BOOL;
	ParametersArray : ParametersArray;
	CommandExternal : TFCommandExternal;
	Timer : REAL := 1;
	Timeout : REAL := 1;
	i : UINT;
	w : UINT;
	e : UINT;
	j : UINT;
	k : UINT;
	z : INT;
	Step : BOOL;
	Power : UINT;
	TimerWorkFlow : ARRAY[0..MAXWORKFLOW] OF REAL;
	WorkFlow : ARRAY[0..MAXWORKFLOW] OF WorkFlow;
	WorkFlowErrorLog : ARRAY[0..MAXWORKFLOW] OF WorkFlowErrorLog;
	NumeroWF : UINT;//Numero del WorkFlow
	
	
	MAN_Actuator : UINT;
	MAN_Cmd : UINT;
	Timer1000 : REAL := 1;
	HornClock : BOOL;
	HornAck : BOOL;
	
	LGVPhaseStopRequest : BOOL;
	//LoopFlipFlop : BOOL;
	//LFF_X : LREAL;
	//LFF_Y : LREAL;
	//LFF_Z : LREAL;
	//LFF_J : LREAL;
	
	ExternalWaitPositionRequest : BOOL;
	//ValidationResult : INT;
	//NextCommand : INT;
	//NextCode : INT;
	AirAlarmTrig : BOOL;
	Volt24Trig : BOOL;
	BeltSafetyTRIG : BOOL;
	//RADIUS : LREAL;
	ClockLamp : BOOL;
	TimerLamp : REAL := 1;
	TimerComTrasporti : REAL :=1;
	AutoTrig : BOOL;
	AutoToMan : BOOL;
	GateAccesTrig : BOOL;
	GateAcces : BOOL;
	ExecuteStopTilter : BOOL;
	ExecuteStopTilterTRIG : BOOL;
	
	TFPalletizerWorkAreaManagerTF 	: TFPalletizerWorkAreaManagerTF_Lastre;
	TFProgramma_Ciclo_Riposo 		: TFProgramma_Ciclo_Riposo_Lastre;
	TFProgramma_Ciclo_Falda 		: TFProgramma_Ciclo_Falda_Lastre;
	TFProgramma_Ciclo_Lastra 		: TFProgramma_Ciclo_Lastra;
	
	(* Ciclo di lavoro CON interpolazione degli assi *)
	TFCiclo_Di_Riposo 				: TFCiclo_Di_Riposo_Lastre;
	TFCiclo_Prelievo_Falda 			: TFCiclo_Prelievo_Falda;
	TFCiclo_Deposito_Falda 			: TFCiclo_Deposito_Falda;
	TFCiclo_Prelievo_Lastra 		: TFCiclo_Prelievo_Lastra;
	TFCiclo_Deposito_Lastra 		: TFCiclo_Deposito_Lastra;
	//Depalettizzatore	
	//TFCiclo_Prelievo_Lastra_Depalettizzatore 		: TFCiclo_Prelievo_Lastra_Depal;
	TFCiclo_Prelievo_Lastra_Depalettizzatore 		: TFCiclo_Prelievo_Lastra_Depal;//TFCiclo_Prelievo_Lastra;
	TFCiclo_Deposito_Lastra_Depalettizzatore 		: TFCiclo_Deposito_Lastra_Depal;
	TFCiclo_Deposito_Falda_Depalettizzatore 		: TFCiclo_Deposito_Falda_Depal;
	
	(* FB Vari *)
	TFCalcoloTraiettoria 				: TFCalcoloTraiettoriaLastre;// TFCalcoloTraiettoria;
	TFCalcoliFuoriIngombri		 		: TFCalcoliFuoriIngombri;
	TFCalcoloPuntiDiAnticipoDinamici 	: TFCalcoloPuntiDiAnticipoDinamici;
	TFValutaAssiInFinestraDiPassMode 	: TFValutaAssiInFinestraDiPassMode;
	
	AbilitazioCiclo_TEST_STEP 	: BOOL := FALSE; 		//TRUE se in fase di test si vuole eseguire il ciclo a step
	CommandSTEP				: BOOL := FALSE;	 //Comando di step per eseguire il ciclo a step

	CommandSTEPTRIG			: BOOL := FALSE;	// Memoria Comando di step per eseguire il ciclo a step
	STEPCicloDONE 			: BOOL;
	PX_GripPresenceOK       : BOOL;
	ErroreDiInterferenza : UINT;
	WaitPositionRequest : BOOL;
	InWaitPosition : BOOL;
	//DepositoFaldaSuCatastaVuoti : BOOL;
	//Filtro_PX_GripPresence : Signal_Filter;
	PX_GripPresenceFiltrata	: BOOL;
	
	PalletLayerPresence : UINT;
	DepositoPaccoInLenta : BOOL;
	
	//CoppiaPinzaOK : BOOL;
	//TimerControlloCoppiaTRUE : REAL;
	//TimerControlloCoppiaFALSE : REAL;
	//FiltroControlloCoppia : REAL := 200;
	
	ForzaPrelievoPaccoDuranteCicloDiRiposo : BOOL;
	
	TimerPacchi1Minuto : REAL;
	AttivaTimerContaPacchi1Minuto : BOOL;
	AttivaTimerContaPacchi5Minuti : BOOL;
	PacchiPrelevatiIn5MinutiAppoggio : REAL;
	cuontpac : UINT;
	Pacchi1Minuto : uint;
	TimerDone1 : UINT;
	TimerPacchi5Minuti : REAL;
	//RibaltinoPronto : BOOL;
	//RichiestaStartRibaltino : BOOL;
	ResetComandoRibaltinoEseguito : BOOL;
	
	//UltimaWaDepositoPacco : INT;
	//UltimoComandoRibaltino : INT;
	//PHOKDebug : bool;
	//CoppiaOkDebug : BOOL;
	Interpolazione_Assi : TFInterpolazioneAssi.Interpolazione_Assi;
	IndiceForSb : int;
	PinzaInQuotaFuoriIngombro : BOOL;// la Quota della pinza mi garantisce che sono in fuori ingombro

	RitardoEsecuzioneInterpolazione : REAL := 0.008;
	TempoCompensazioneDecelerazione : REAL := 0.03;
	TempoCompensazioneAccelerazione : REAL := 0;
	
	TimerRestCmdRibaltino : REAL;
	
	//ComandoPickPoint : ARRAY[1..10] OF INT;
	//StatoPickPoint : ARRAY[1..10] OF INT;
	//comdRib : INT :=1;
	wfindx : UINT;
	PinzaConProdottoInPresa : BOOL;
	
	TimerONAlternato : REAL;
	TimerOFFAlternato : REAL;
	TimerSirenaOFF_Segnalazioni : REAL;
	In_GiCavallete: UINT;
	OkEstacionFinPiking: BOOL;
END_VAR

(* Init *)
IF NOT Init THEN
	TFCommandBufferClear(ADR(Cmd));
	TFCommandClear(ADR(CmdNext));
	TFCommandExeClear(ADR(CmdExe));
	TFStateUpdate(ADR(State),StateNOP);
	TFErrorClear(ADR(Error));
	TFWarningClear(ADR(Warning));
	OUT.HomeDone := FALSE;
	AutoToMan := TRUE;
	Timer := 10;
	Timeout := 10;
	OUT.PowerOffTilterReq := FALSE;
	OUT.StopTilterReq := FALSE;
	OUT.PowerOnTilterReq := FALSE;
	OUT.ResetTilterReq := FALSE;
	OUT.StartTilter := FALSE;
	Init := TRUE;
END_IF
PosRobot := 0 ;
RobotWorkAreaCavallete := FALSE ;

IF NuEstacionesPiking > 1  THEN
	MultiplesCavalletesReceta := TRUE ;
ELSE
	MultiplesCavalletesReceta := FALSE ;
END_IF

IF NuEstacionesPiking > 1 AND NuEstacionPiking <> 0 AND WorkAreaState^[NuEstacionPiking].Supporto.Tipologia = CAVALLETTO THEN
	PikingConCavallete := TRUE ;
ELSE
	PikingConCavallete := FALSE ;
END_IF


 
(*IF MultiplesCavalletesReceta THEN 
	IF NuEstacionPiking = 1  THEN 
		NuPosGuiroPiking := NuEstacionPiking + 1 ;
	ELSIF NuEstacionPiking > 1 AND NuEstacionesPiking <  NuEstacionPiking      THEN  
		NuPosGuiroPiking := NuEstacionPiking - 1 ;
	END_IF
	
END_IF *)

WaCavalleteEnPiking := 0 ;
IF MultiplesCavalletesReceta THEN 
	FOR In_GiCavallete := 1 TO MAXAREAPRESENT DO 
		IF PosCavalleteOrdenPikin[In_GiCavallete] = CAVALLETTO THEN
			IF In_GiCavallete = NuEstacionPiking AND In_GiCavallete = 1   THEN
				NuPosGuiroPiking := NuEstacionPiking + 1 ;
			ELSIF  In_GiCavallete = NuEstacionPiking   THEN  
				IF WaCavalleteEnPiking = 0 THEN 
					NuPosGuiroPiking := NuEstacionPiking + 1 ;
					ELSE
					NuPosGuiroPiking := NuEstacionPiking - 1 ;	
				END_IF
			ELSIF  In_GiCavallete <> NuEstacionPiking   THEN  
				WaCavalleteEnPiking := WaCavalleteEnPiking +1 ;	
			END_IF
				
		END_IF
	END_FOR
END_IF

IF NOT MultiplesCavalletesReceta AND  NuEstacionPiking <> 0 AND 
					WorkAreaState^[NuEstacionPiking].Supporto.Tipologia = CAVALLETTO AND
							 PosFinOrdenPikingCaballete = 0  THEN 
	OkEstacionFinPiking := FALSE ;
	CASE NuEstacionPiking OF
		1 :
			FOR In_GiCavallete := (NuEstacionPiking +1) TO MAXAREAPRESENT DO
				IF WorkAreaState^[In_GiCavallete].Supporto.Tipologia <> CAVALLETTO THEN
					PosFinOrdenPikingCaballete := In_GiCavallete ;
					EXIT ;
				END_IF
			END_FOR
			
		2..20 :
			
			FOR In_GiCavallete := (NuEstacionPiking-1)  TO 1 BY -1 DO
				IF WorkAreaState^[In_GiCavallete].Supporto.Tipologia <> CAVALLETTO THEN
					PosFinOrdenPikingCaballete := In_GiCavallete ;
					OkEstacionFinPiking := TRUE ;
					EXIT ;
				END_IF
			END_FOR	
			IF NOT OkEstacionFinPiking THEN 
				FOR In_GiCavallete := (NuEstacionPiking +1)  TO MAXAREAPRESENT  DO
				IF WorkAreaState^[In_GiCavallete].Supporto.Tipologia <> CAVALLETTO THEN
					PosFinOrdenPikingCaballete := In_GiCavallete ;
					OkEstacionFinPiking := TRUE ;
					EXIT ;
				END_IF
			END_FOR	
			END_IF
			
	END_CASE

	ELSE 
		
		IF NuPosGuiroPiking <> 0 THEN 
			PosFinOrdenPikingCaballete := NuPosGuiroPiking ; 
		END_IF
END_IF


FOR In_PosRobot := 1 TO MAXAREAPRESENT DO
	IF TFAsseInFinestra(Posizione_Attuale:= Modules^.AX_X.Ax^.AxRef^.NcToPlc.ActPos ,Posizione_Finale:= WorkArea^[In_PosRobot].X ,FinestraDiControllo := 300) THEN
		PosRobot := In_PosRobot ;
		RobotCentroPosX := TRUE ;	
			IF WorkAreaState^[PosRobot].Supporto.Tipologia = CAVALLETTO THEN
				RobotWorkAreaCavallete := TRUE ;
				
			ELSE
				RobotWorkAreaCavallete := False ;	
			END_IF
		
		 	IF 	 Modules^.AX_J.Ax^.AxRef^.NcToPlc.ActPos <85 THEN 
					PosicionJActual := 0 ;
				ELSIF Modules^.AX_J.Ax^.AxRef^.NcToPlc.ActPos >95 THEN
					 PosicionJActual := 180 ;
				ELSE
					PosicionJActual := 90 ;
				END_IF
		EXIT;
		ELSE
		RobotCentroPosX := FALSE ;		
		
	END_IF
END_FOR 

IF RobotCentroPosX THEN 
	EjexEnPosicion  := WorkArea^[PosRobot].X ;
	ELSE
	EjexEnPosicion := 0;	
	
END_IF


IF 	 Mission^.JPlace <85 THEN 
	PosicionJDestino := 0 ;
ELSIF Mission^.JPlace >95 THEN
	 PosicionJDestino := 180 ;
ELSE
	PosicionJDestino := 90 ;
END_IF
IF 	 Mission^.JPick <85 THEN 
	PosicionJOrigen := 0 ;
ELSIF Mission^.JPick >95 THEN
	 PosicionJOrigen := 180 ;
ELSE
	PosicionJOrigen := 90 ;
END_IF

IF PosicionJDestino <> PosicionJOrigen  OR PosicionJActual <> PosicionJOrigen THEN 
	AngulosDiferentes := TRUE ;
	ELSE 
	AngulosDiferentes := FALSE ;	
END_IF





AbilitazioCiclo_TEST_STEP := HMI_AbilitazioneCicloAStep;
CommandSTEP := HMI_CommandSTEP OR (AbilitazioCiclo_TEST_STEP AND IN.Mode.ResetRequest);

(* Generic Timer - Add here all your Timers *)

TFTimerCall(ADR(Timer),Cfg.TimeBase);
TFTimerCall(ADR(Timeout),Cfg.TimeBase);
TFTimerCall(ADR(Timer1000),Cfg.TimeBase);
TFTimerCall(ADR(TimerWorkFlow[0]),Cfg.TimeBase);
TFTimerCall(ADR(TimerWorkFlow[1]),Cfg.TimeBase);
TFTimerCall(ADR(TimerWorkFlow[2]),Cfg.TimeBase);
TFTimerCall(ADR(TimerWorkFlow[3]),Cfg.TimeBase);
TFTimerCall(ADR(TimerWorkFlow[4]),Cfg.TimeBase);
TFTimerCall(ADR(TimerWorkFlow[5]),Cfg.TimeBase);
TFTimerCall(ADR(TimerWorkFlow[6]),Cfg.TimeBase);
TFTimerCall(ADR(TimerWorkFlow[7]),Cfg.TimeBase);
TFTimerCall(ADR(TimerWorkFlow[8]),Cfg.TimeBase);
TFTimerCall(ADR(TimerLamp),Cfg.TimeBase);
//TFTimerCall(ADR(TimerControlloCoppiaTRUE),Cfg.TimeBase);
//TFTimerCall(ADR(TimerControlloCoppiaFALSE),Cfg.TimeBase);
TFTimerCall(ADR(TimerComTrasporti),Cfg.TimeBase);
TFTimerCall(ADR(TimerRestCmdRibaltino),Cfg.TimeBase);

(* External Command *)
CommandExternal(
	Cmd := ADR(Cmd),
	CmdExe := ADR(CmdExe),
	State := ADR(state),
	Error := ADR(Error),
	ErrorLog := ADR(ErrorLog),
	Warning := ADR(Warning),
	WarningLog := ADR(WarningLog),
	Mode := ADR(IN.Mode));

(* External To Buffered Command *)
TFCommandToNext(ADR(Cmd),ADR(CmdNext),ADR(CmdExe),ADR(Cfg),ADR(Error),ADR(ErrorLog),ADR(State));

(* Buffered To Exe Command *)
TFCommandToExecution(ADR(CmdNext),ADR(CmdExe),ADR(Error),ADR(ErrorLog),ADR(State),ADR(CmdLog));

(* Exe Command *)
CASE CmdExe.Code OF

	(* ******************************************************************************************************** *)
	(* Nop *)
	(* ******************************************************************************************************** *)
	CmdNOP:	;

	(* ******************************************************************************************************** *)
	(* Stop *)
	(* ******************************************************************************************************** *)
	CmdSTOP:
		CASE CmdExe.CmdCase OF
			(* Case 0 *)
			0: 	TFStateUpdate(ADR(State),StateSTOP_RUN);
				TFTimerSet(ADR(Timer),10,TRUE);
				TFTimerSet(ADR(Timeout),5000,TRUE);
				OUT.StartHorn := FALSE;
				OUT.PowerOffTilterReq := FALSE;
				OUT.StopTilterReq := FALSE;
				OUT.PowerOnTilterReq := FALSE;
				OUT.ResetTilterReq := FALSE;
				OUT.StartTilter := FALSE;
				TFCommandCase(ADR(CmdExe),1,CommandCase_INC);
			
			(* Case 1 - Wait All WorkFlow=FALSE *)
			1:	IF (*NOT WorkFlow[0].Enable AND
					NOT WorkFlow[1].Enable AND
					NOT WorkFlow[2].Enable AND
					NOT WorkFlow[3].Enable AND
					NOT WorkFlow[4].Enable AND
					NOT WorkFlow[5].Enable AND
					NOT WorkFlow[6].Enable AND
					NOT WorkFlow[7].Enable AND
					NOT WorkFlow[8].Enable*)
					TFWorkflowsAllEnableOrDisable(ADR(WorkFlow),FALSE) OR
					TFTimerDone(ADR(Timer)) THEN
					TFCommandCase(ADR(CmdExe),1,CommandCase_INC);
				END_IF
			
			(* Case 2 - Invio comando di STOP a tuttti i moduli *)
			2:	//OUT.HomeDone := FALSE;
				//Disabilito tutti i WF				
				FOR wfindx := 0 TO MAXWORKFLOW DO
					WorkFlow[wfindx].Enable := FALSE;
				END_FOR
				TFParametersArrayClear(ADR (ParametersArray));
				TFPalletizerModulesCommandSend(CmdSTOP,ParametersArray,Modules);
				OUT.StopTilterReq := ExecuteStopTilter;
				TFCommandCase(ADR(CmdExe),1,CommandCase_INC);

			(* Case 3 - Attesa che tutti i moduli abbiano completato il comando *)
			3:	IF TFPalletizerModulesCheckState(StateSTOP_END,Modules) THEN
					TFCommandCase(ADR(CmdExe),100,CommandCase_JMP);
				ELSIF TFTimerDone(ADR(Timeout)) THEN
					TFError(ErrTOSTOP,ErrNULL,ADR(CmdExe),ADR(State),ADR(Error),ADR(ErrorLog));
				END_IF

			(* Case 100 *)
			100:TFStateUpdate(ADR(State),StateSTOP_END);
				TFCommandExeClear(ADR(CmdExe));

			ELSE
				TFError(ErrNOCMDCASE,ErrNULL,ADR(CmdExe),ADR(State),ADR(Error),ADR(ErrorLog));
		END_CASE
	
	(* ******************************************************************************************************** *)
	(* Error Reset *)
	(* ******************************************************************************************************** *)
	CmdRESET:
		CASE CmdExe.CmdCase OF
			(* Case 0 *)
			0: 	TFStateUpdate(ADR(State),StateRESET_RUN);
				TFTimerSet(ADR(Timeout),1000,TRUE);
				OUT.StartHorn := FALSE;
				AirAlarmTrig := FALSE;
				Volt24Trig  := FALSE;
				BeltSafetyTRIG := FALSE;
				PalletStackEmpty := 0;
				LayerStackEmpty := 0;
				(* Se l'errore di interferenza è maggiore di 0, assegno alla traiettoria e alla missione dei i valori del punto di riposo, 
				in questo modo sbianco le eventuali quote non ammesse *)
				IF ErroreDiInterferenza > 0 THEN
					//X_Riposo	:= WorkPickPoint^[1].Xv;
					//Y_Riposo	:= WorkPickPoint^[1].Yv;
					//Z_Riposo	:= ZRESTPOSITION;
					//J_Riposo	:= WorkPickPoint^[1].Jv;
					//K_Riposo	:= KRESTPOSITION; 
					
					{info 'TODO: Valorizzar quote di riposo'} 
					Traiettoria^.EndPoint.X := X_Riposo;
					Traiettoria^.EndPoint.Y := Y_Riposo;
					Traiettoria^.EndPoint.Z := Z_Riposo;
					Traiettoria^.EndPoint.J := J_Riposo;
					Traiettoria^.EndPoint.K := K_Riposo;
					
					Mission^.PPick			:= PICKPOINT1;
					Mission^.TPick 			:= TPICK_NOT_DEFINED;
					Mission^.XPick 			:= X_Riposo;
					Mission^.YPick 			:= Y_Riposo;
					Mission^.ZPick 			:= Z_Riposo;
					Mission^.JPick 			:= J_Riposo;
					
					Mission^.XPlace := X_Riposo;
					Mission^.YPlace := Y_Riposo;
					Mission^.ZPlace := Z_Riposo;
					Mission^.JPlace := J_Riposo;
					
					ErroreDiInterferenza := 0;
				END_IF
							
				
				LGVError := 0;
				GateAccessError := 0;
				TFCommandCase(ADR(CmdExe),1,CommandCase_INC);

			(* Case 1 - Invio comando di reset a tuttti i moduli*)
			1:	TFParametersArrayClear(ADR (ParametersArray));
				TFPalletizerModulesCommandSend(CmdRESET,ParametersArray,Modules);
				TFCommandCase(ADR(CmdExe),1,CommandCase_INC);

			(* Case 2 - Attesa che tutti i moduli abbiano completato il comando *)
			2:	
				IF TFPalletizerModulesCheckState(StateRESET_END,Modules) THEN
						TFCommandCase(ADR(CmdExe),99,CommandCase_JMP);
				ELSIF TFTimerDone(ADR(Timeout)) THEN
					OUT.ResetTilterReq := FALSE;
					TFError(ErrTORESET,ErrNULL,ADR(CmdExe),ADR(State),ADR(Error),ADR(ErrorLog));
				END_IF

			(* Case 99 *)
			99:	
				FOR i:= 0 TO MAXWORKFLOW DO
					IF WorkFlow[i].WFCase = StateWF_ERROR THEN
						WorkFlow[i].WFCase := 0;
					END_IF
					IF WorkFlow[i].State = StateWF_ERROR THEN
						WorkFlow[i].State := 0;
					END_IF
				END_FOR
				TFErrorClear(ADR(Error));
				TFWarningClear(ADR(Warning));
				TFCommandCase(ADR(CmdExe),100,CommandCase_JMP);
				
			(* Case 100 *)
			100:TFStateUpdate(ADR(State),StateRESET_END);
				TFCommandExeClear(ADR(CmdExe));

			ELSE
				TFError(ErrNOCMDCASE,ErrNULL,ADR(CmdExe),ADR(State),ADR(Error),ADR(ErrorLog));
		END_CASE

	(* ******************************************************************************************************** *)
	(* Power *)
	(* ******************************************************************************************************** *)
	CmdPOWER:
		CASE CmdExe.CmdCase OF
			(* Case 0 *)
			0: 	TFStateUpdate(ADR(State),StatePOWER_RUN);
				TFTimerSet(ADR(Timeout),2500,TRUE);

				IF TFCommandParRead(CmdExe.Cmd.Parameter,ADR(ParametersArray),1) THEN
					Power := STRING_TO_UINT(ParametersArray.Parameters[0]);
				ELSE
					TFError(ErrCMDPARNUM,ErrNULL,ADR(CmdExe),ADR(State),ADR(Error),ADR(ErrorLog));
					RETURN;
				END_IF

				IF Power = 1 THEN
					TFCommandCase(ADR(CmdExe),10,CommandCase_JMP);
				ELSE
					TFCommandCase(ADR(CmdExe),20,CommandCase_JMP);
				END_IF
				
			(* Case 10 - Power On *)
			10: OUT.PowerActive := TRUE;
				OUT.PowerActiveSIMULAZIONE := FALSE;
				IF IN.PowerOk THEN
					TFCommandCase(ADR(CmdExe),1,CommandCase_INC);
				ELSIF TFTimerDone(ADR(Timeout)) THEN
					OUT.PowerActive := FALSE;
					TFError(ErrTOPOWERON,ErrNULL,ADR(CmdExe),ADR(State),ADR(Error),ADR(ErrorLog));
				END_IF
			
			(* Case 11 - Invio comando di Power *)
			11:	TFParametersArrayClear(ADR (ParametersArray));
				ParametersArray.Parameters[0] := '1';
				TFPalletizerModulesCommandSend(CmdPOWER,ParametersArray,Modules);
				TFCommandCase(ADR(CmdExe),1,CommandCase_INC);
			
			(* Case 12 - Attesa che tutti i moduli siano in Power *)
			12:IF TFPalletizerModulesCheckState(StatePOWER_END,Modules) THEN
					TFCommandCase(ADR(CmdExe),100,CommandCase_JMP);
				ELSIF TFPalletizerIsModuleError(Modules) THEN
					OUT.PowerActive := FALSE;
					TFError(ErrNOPOWER,ErrNULL,ADR(CmdExe),ADR(State),ADR(Error),ADR(ErrorLog));
				ELSIF TFTimerDone(ADR(Timeout)) THEN
					OUT.PowerActive := FALSE;
					TFError(ErrTOPOWERON,ErrNULL,ADR(CmdExe),ADR(State),ADR(Error),ADR(ErrorLog));
				END_IF
			
			(* Case 20 - Power Off *)
			20:	CmdExe.RapidStopRequest := 1;
				CmdExe.PhaseStopRequest := 1;
				TFCommandCase(ADR(CmdExe),1,CommandCase_INC);
			
			(* Case 21 *)
			21:					
				//Disabilito tutti i WF				
				FOR wfindx := 0 TO MAXWORKFLOW DO
					WorkFlow[wfindx].Enable := FALSE;
				END_FOR

				TFParametersArrayClear(ADR (ParametersArray));
				TFPalletizerModulesCommandSend(CmdSTOP,ParametersArray,Modules);
				TFCommandCase(ADR(CmdExe),1,CommandCase_INC);
			
			(* Case 22 *)
			22: IF TFPalletizerModulesCheckState(StateSTOP_END,Modules) THEN
					TFCommandCase(ADR(CmdExe),1,CommandCase_INC);
				ELSIF TFTimerDone(ADR(Timeout)) THEN
					TFError(ErrTOSTOP,ErrNULL,ADR(CmdExe),ADR(State),ADR(Error),ADR(ErrorLog));
				END_IF

			(* Case 23 *)
			23:	TFParametersArrayClear(ADR (ParametersArray));
				ParametersArray.Parameters[0] := '0';
				TFPalletizerModulesCommandSend(CmdPOWER,ParametersArray,Modules);
				TFCommandCase(ADR(CmdExe),1,CommandCase_INC);
			
			(* Case 24 *)
			24:	IF TFPalletizerModulesCheckState(StatePOWER_END,Modules) THEN
					OUT.PowerActive := FALSE;
					OUT.PowerOffTilterReq := FALSE;
					OUT.PowerActiveSIMULAZIONE := FALSE;
					TFCommandCase(ADR(CmdExe),1,CommandCase_INC);
				ELSIF TFPalletizerIsModuleError(Modules) THEN
					OUT.PowerActive := FALSE;
					TFError(ErrNOPOWER,ErrNULL,ADR(CmdExe),ADR(State),ADR(Error),ADR(ErrorLog));
				ELSIF TFTimerDone(ADR(Timeout)) THEN
					OUT.PowerOffTilterReq := FALSE;
					OUT.PowerActive := FALSE;
					TFError(ErrTOPOWEROFF,ErrNULL,ADR(CmdExe),ADR(State),ADR(Error),ADR(ErrorLog));
				END_IF
				
			(* Case 25 - Power On *)
			25: OUT.PowerActive := FALSE;
				IF NOT IN.PowerOk THEN
					TFCommandCase(ADR(CmdExe),100,CommandCase_JMP);
				ELSIF TFTimerDone(ADR(Timeout)) THEN
					OUT.PowerActive := FALSE;
					TFError(ErrTOPOWEROFF,ErrNULL,ADR(CmdExe),ADR(State),ADR(Error),ADR(ErrorLog));
				END_IF

			(* Case 100 *)
			100:TFStateUpdate(ADR(State),StatePOWER_END);
				TFCommandExeClear(ADR(CmdExe));

			ELSE
				TFError(ErrNOCMDCASE,ErrNULL,ADR(CmdExe),ADR(State),ADR(Error),ADR(ErrorLog));
		END_CASE
	
	(* ******************************************************************************************************** *)
	(* Home *)
	(* ******************************************************************************************************** *)
	CmdHOME:
		CASE CmdExe.CmdCase OF
			(* Case 0 *)
			0: 	TFStateUpdate(ADR(State),StateHOME_RUN);
				TFTimerSet(ADR(Timeout),60000,TRUE);
				OUT.HomeDone := FALSE;
				TFCommandCase(ADR(CmdExe),10,CommandCase_JMP);

			(* Case 10 *)
			10:	TFCommandCase(ADR(CmdExe),1,CommandCase_INC);

				(* Check Modules Error *)
				IF TFPalletizerIsModuleError(Modules) THEN
					TFCommandCase(ADR(CmdExe),100,CommandCase_JMP);
				END_IF

			(* Case 11 - Start Horn *)
			11:	TFTimerSet(ADR(Timer),1000,NOT OUT.StartHorn);
				OUT.StartHorn := TRUE;
				IF TFTimerDone(ADR(Timer)) THEN
					OUT.StartHorn := FALSE;
					TFCommandCase(ADR(CmdExe),1,CommandCase_INC);
				END_IF
				IF CmdExe.PhaseStopRequest > 0 THEN
					OUT.StartHorn := FALSE;
					TFCommandCase(ADR(CmdExe),100,CommandCase_JMP);
				END_IF

			(* Case 12 - Homing *)
			12:	WorkFlow[0].Enable := TRUE;
				TFWorkFlowCase(ADR(WorkFlow[0]),0,WorkflowCase_JMP);
				TFCommandCase(ADR(CmdExe),1,CommandCase_INC);

			(* Case 13 - Wait Homing END *)
			13:	IF WorkFlow[0].State = StateWF_END THEN
					TFCommandCase(ADR(CmdExe),100,CommandCase_JMP);
				ELSIF WorkFlow[0].WFCase = StateWF_ERROR THEN
					WorkFlow[0].Enable := FALSE;
					TFError(ErrWF,ErrNULL,ADR(CmdExe),ADR(State),ADR(Error),ADR(ErrorLog));
				END_IF

			(* Case 100 *)
			100:TFStateUpdate(ADR(State),StateHOME_END);
				TFCommandExeClear(ADR(CmdExe));

			ELSE
				TFError(ErrNOCMDCASE,ErrNULL,ADR(CmdExe),ADR(State),ADR(Error),ADR(ErrorLog));
		END_CASE


	(* ******************************************************************************************************** *)
	(* Manual *)
	(* ******************************************************************************************************** *)
	CmdMAN:
		CASE CmdExe.CmdCase OF
			(* Case 0 *)
			0: 	TFStateUpdate(ADR(State),StateMAN_RUN);
				TFTimerSet(ADR(Timeout),10,TRUE);
				//OUT.HomeDone := FALSE;
				IF TFCommandParRead(CmdExe.Cmd.Parameter,ADR(ParametersArray),2) THEN
					MAN_Actuator	:= STRING_TO_UINT(ParametersArray.Parameters[0]);
					MAN_Cmd		:= STRING_TO_UINT(ParametersArray.Parameters[1]);
				ELSE
					TFError(ErrCMDPARNUM,ErrNULL,ADR(CmdExe),ADR(State),ADR(Error),ADR(ErrorLog));
					RETURN;
				END_IF

				CASE MAN_Actuator OF
					(* Case 0..99 for Actuators *)
					(* Case 100..199  for Axis *)
					(* Case 200.....  for Modules *)

					(* Case Nop *)
					0: 	;

					(* Case 1:  *)
					1:	CASE MAN_Cmd OF
							0:	;
							
							ELSE
								TFError(ErrNOCMDCASE,ErrNULL,ADR(CmdExe),ADR(State),ADR(Error),ADR(ErrorLog));
						END_CASE;

					(* Case 200:  Module Robot *)
					200:CASE MAN_Cmd OF
							0:	;
							
							
							1: 
								TFCommandCase(ADR(CmdExe),1000,CommandCase_JMP);
							ELSE
								TFError(ErrNOCMDCASE,ErrNULL,ADR(CmdExe),ADR(State),ADR(Error),ADR(ErrorLog));
						END_CASE;

					ELSE
						TFError(ErrNOCMDCASE,ErrNULL,ADR(CmdExe),ADR(State),ADR(Error),ADR(ErrorLog));
				END_CASE

				IF CmdExe.CmdCase = 0 THEN
					TFCommandCase(ADR(CmdExe),1,CommandCase_INC);
				END_IF

			(* Case 1 *)
			1: 	IF (MAN_Cmd = 0) OR TFTimerDone(ADR(Timeout)) THEN
					(* Clear All Output Here *)
					TFCommandCase(ADR(CmdExe),100,CommandCase_JMP);
					TFCommandExeClear(ADR(CmdExe));
				END_IF
			
			(* *)	
			201:
				
				TFCommandCase(ADR(CmdExe),1000,CommandCase_JMP);
			
			(* Case 1000 *)
			1000:
				TFStateUpdate(ADR(State),StateMAN_END);
				TFCommandExeClear(ADR(CmdExe));
			
			ELSE
				TFError(ErrNOCMDCASE,ErrNULL,ADR(CmdExe),ADR(State),ADR(Error),ADR(ErrorLog));
		END_CASE;


	CmdCICLORIPOSO:	
		CASE CmdExe.CmdCase OF

			(* Case 0 *)
			0: 	TFStateUpdate(ADR(State),StateCICLORIPOSO_RUN);
				TFCommandCase(ADR(CmdExe),10,CommandCase_JMP);

			(* Case 10 *)
			10:	TFCommandCase(ADR(CmdExe),1,CommandCase_INC);
				
				(* Check Modules Power *)
				IF NOT IN.PowerOk OR NOT TFPalletizerModulesCheckPowerActive(Modules) THEN
					TFError(ErrMACHINEPALLETIZER_MISSINGPOWER,ErrNULL,ADR(CmdExe),ADR(State),ADR(Error),ADR(ErrorLog));
				END_IF

				(* Check Modules Error *)
				IF TFPalletizerIsModuleError(Modules) THEN
					TFCommandCase(ADR(CmdExe),100,CommandCase_JMP);
				END_IF

			(* Case 11 - Start Horn *)
			11:	TFTimerSet(ADR(Timer),3000,NOT OUT.StartHorn);
				OUT.StartHorn := TRUE;
				IF TFTimerDone(ADR(Timer)) THEN
					OUT.StartHorn := FALSE;
					TFCommandCase(ADR(CmdExe),14,CommandCase_JMP);
				END_IF
				IF CmdExe.RapidStopRequest > 0 OR
					CmdExe.PhaseStopRequest > 0 THEN
					OUT.StartHorn := FALSE;
					TFCommandCase(ADR(CmdExe),100,CommandCase_JMP);
				END_IF;

			(* Case 14 - Attivazione e inizializzazione del Workflow*)
			14:	WorkFlow[2].Enable := TRUE;
				TFWorkFlowCase(ADR(WorkFlow[2]),0,WorkflowCase_JMP);
				TFCommandCase(ADR(CmdExe),1,CommandCase_INC);

			(* Case 15 - Attesa di un eventuale stop rapido/stop in fase o attesa del completamento/errore workflow *)
			15:	IF CmdExe.RapidStopRequest > 0 OR
					CmdExe.PhaseStopRequest > 0 OR
					(NOT WorkFlow[2].Enable OR WorkFlow[2].WFCase = StateWF_ERROR) THEN
					TFCommandCase(ADR(CmdExe),1,CommandCase_INC);
				END_IF;

			(* Case 16 - Wait WF End *)
			16: IF (NOT WorkFlow[2].Enable OR WorkFlow[2].State = StateWF_END OR WorkFlow[2].WFCase = StateWF_ERROR) THEN
				WorkFlow[2].Enable := FALSE;
				IF WorkFlow[2].WFCase = StateWF_ERROR THEN
					IF Warning.Code <> ErrNULL THEN
						TFError(Warning.Code,ErrNULL,ADR(CmdExe),ADR(State),ADR(Error),ADR(ErrorLog));
					ELSE
						TFError(ErrWF,ErrNULL,ADR(CmdExe),ADR(State),ADR(Error),ADR(ErrorLog));
					END_IF
				ELSE
					(*Invio comando di stop ai moduli*)
					TFParametersArrayClear(ADR (ParametersArray));
					TFPalletizerModulesCommandSend(CmdSTOP,ParametersArray,Modules);
					IF TFIsModuleWarning(Warning) THEN
						TFError(Warning.Code,ErrNULL,ADR(CmdExe),ADR(State),ADR(Error),ADR(ErrorLog));
					ELSE
						TFCommandCase(ADR(CmdExe),100,CommandCase_JMP);
					END_IF
				END_IF
			END_IF	

			(* End Case *)
			100:TFStateUpdate(ADR(State),StateCICLORIPOSO_END);
				TFCommandExeClear(ADR(CmdExe));

			ELSE
				TFError(ErrNOCMDCASE,ErrNULL,ADR(CmdExe),ADR(State),ADR(Error),ADR(ErrorLog));
		END_CASE

	(* ******************************************************************************************************** *)
	(* DO *)
	(* ******************************************************************************************************** *)
	CmdDO:
		CASE CmdExe.CmdCase OF

			(* Case 0 *)
			0: 	TFStateUpdate(ADR(State),StateDO_RUN);
				TFCommandCase(ADR(CmdExe),10,CommandCase_JMP);

			(* Case 10 *)
			10:	TFCommandCase(ADR(CmdExe),1,CommandCase_INC);
				
				(* Check Modules Power *)
				IF NOT IN.PowerOk OR NOT TFPalletizerModulesCheckPowerActive(Modules) THEN
					TFError(ErrMACHINEPALLETIZER_MISSINGPOWER,ErrNULL,ADR(CmdExe),ADR(State),ADR(Error),ADR(ErrorLog));
				END_IF

				(* Check Modules Error *)
				IF TFPalletizerIsModuleError(Modules) THEN
					TFCommandCase(ADR(CmdExe),100,CommandCase_JMP);
				END_IF

			(* Case 11 - Start Horn *)
			11:	TFTimerSet(ADR(Timer),3000,NOT OUT.StartHorn);
				OUT.StartHorn := TRUE;
				IF TFTimerDone(ADR(Timer)) THEN
					OUT.StartHorn := FALSE;
					TFCommandCase(ADR(CmdExe),1,CommandCase_INC);
				END_IF
				IF CmdExe.PhaseStopRequest > 0 THEN
					OUT.StartHorn := FALSE;
					TFCommandCase(ADR(CmdExe),100,CommandCase_JMP);
				END_IF;

			(* Case 12 - Homing *)
			12:	WorkFlow[0].Enable := TRUE;
				OUT.StartTilter := TRUE;
				TFWorkFlowCase(ADR(WorkFlow[0]),0,WorkflowCase_JMP);
				TFCommandCase(ADR(CmdExe),1,CommandCase_INC);
				
			(* Case 13 - Wait Homing END *)
			13:	IF WorkFlow[0].State = StateWF_END THEN
					IF CmdExe.PhaseStopRequest > 0 THEN
						TFCommandCase(ADR(CmdExe),100,CommandCase_JMP);
					ELSE
						TFCommandCase(ADR(CmdExe),1,CommandCase_INC);
					END_IF
				ELSIF WorkFlow[0].WFCase = StateWF_ERROR THEN
					WorkFlow[0].Enable := FALSE;
					TFError(ErrWF,ErrNULL,ADR(CmdExe),ADR(State),ADR(Error),ADR(ErrorLog));
				END_IF;

			(* Case 14 *)
			14:	WorkFlow[1].Enable := TRUE;
				TFWorkFlowCase(ADR(WorkFlow[1]),0,WorkflowCase_JMP);	
				TFCommandCase(ADR(CmdExe),1,CommandCase_INC);

			(* Case 15 - Wait Stop Request *)
			15:	IF CmdExe.PhaseStopRequest > 0 THEN
					TFCommandCase(ADR(CmdExe),1,CommandCase_INC);
				END_IF;

			(* Case 16 - Wait WF End *)
			16: IF TFIsWorkflowDisableOrEndedOrError(NumWFPresence:=MAXWORKFLOW,ADR(WorkFlow)) THEN //Verifico che tutti i WF non siano attivi, nel caso attendo che lo siano
					//Disabilito tutti i WF				
					FOR wfindx := 0 TO MAXWORKFLOW DO
						WorkFlow[wfindx].Enable := FALSE;
					END_FOR
					
					(*Invio comando di stop ai moduli*)
					TFParametersArrayClear(ADR (ParametersArray));
					TFPalletizerModulesCommandSend(CmdSTOP,ParametersArray,Modules);
	
					IF TFIsWorkflowError(ADR(WorkFlow)) THEN //Valuto se almento un WF è in errore
						IF Warning.Code <> ErrNULL THEN
							TFError(Warning.Code,ErrNULL,ADR(CmdExe),ADR(State),ADR(Error),ADR(ErrorLog));
							TFCommandCase(ADR(CmdExe),100,CommandCase_JMP);
						ELSE
							TFError(ErrWF,ErrNULL,ADR(CmdExe),ADR(State),ADR(Error),ADR(ErrorLog));
							TFCommandCase(ADR(CmdExe),100,CommandCase_JMP);
						END_IF
					ELSE
						IF TFIsModuleWarning(Warning) THEN
							TFError(Warning.Code,ErrNULL,ADR(CmdExe),ADR(State),ADR(Error),ADR(ErrorLog));
							TFCommandCase(ADR(CmdExe),100,CommandCase_JMP);
						ELSE
							TFCommandCase(ADR(CmdExe),100,CommandCase_JMP);
						END_IF
					END_IF
				END_IF	

			(* End Case *)
			100:TFStateUpdate(ADR(State),StateDO_END);
				TFCommandExeClear(ADR(CmdExe));

			ELSE
				TFError(ErrNOCMDCASE,ErrNULL,ADR(CmdExe),ADR(State),ADR(Error),ADR(ErrorLog));
		END_CASE

	ELSE
		TFError(ErrNOCMD,ErrNULL,ADR(CmdExe),ADR(State),ADR(Error),ADR(ErrorLog));	

END_CASE;

(*---------------------------------------------------------*)
(* Descrizione WorkFlow *)
(*---------------------------------------------------------*)
(* 
	-	WF0: WF di Gestione Ciclo di Home
	-	WF1: WF Principale
	-	WF2: WF Ciclo di Riposo
	-	WF3: WF Ciclo Prelievo Pallet
	-	WF4: WF Ciclo Deposito Pallet
	-	WF5: WF Ciclo Prelievo Falda
	-	WF6: WF Ciclo Deposito Falda
	-	WF7: WF Ciclo Prelievo Pacco
	-	WF8: WF Ciclo Deposito Pacco                       *)

(*---------------------------------------------------------*)
(*---------------------------------------------------------*)

(*-------------------------------------------------------------------------------------------*)		
(* WorkFlow 0 - Homing *)
(*-------------------------------------------------------------------------------------------*)
IF WorkFlow[0].Enable THEN

	CASE WorkFlow[0].WFCase OF

		(* Case 0 *)
		0: 	WorkFlow[0].State := StateWF_RUN;
			TFTimerSet(ADR(TimerWorkFlow[0]),2000,TRUE);
			TFWorkFlowCase(ADR(WorkFlow[0]),1,WorkflowCase_INC);

		(* Case 1 *)
		1:	IF CmdExe.RapidStopRequest > 0 OR
				CmdExe.PhaseStopRequest > 0 THEN
				TFWorkFlowCase(ADR(WorkFlow[0]),100,WorkflowCase_JMP);
			ELSE
				(* Check Modules Error *)
				IF TFPalletizerIsModuleError(Modules) THEN
						CmdExe.PhaseStopRequest := 1;
						//OUT.HomeDone := FALSE;
						TFWorkFlowCase(ADR(WorkFlow[0]),StateWF_ERROR,WorkflowCase_JMP);
				ELSE
					IF NOT OUT.HomeDone OR (NOT OUT.HomeDone AND 
						(NOT Modules^.AX_X.Ax^.AxRef^.Status.Homed OR
						NOT Modules^.AX_Y.Ax^.AxRef^.Status.Homed OR
						NOT Modules^.AX_Z.Ax^.AxRef^.Status.Homed OR
						NOT Modules^.AX_J.Ax^.AxRef^.Status.Homed)) THEN
						
							TFWorkFlowCase(ADR(WorkFlow[0]),25,WorkflowCase_JMP);
					ELSE
						OUT.HomeDone := TRUE;
						TFWorkFlowCase(ADR(WorkFlow[0]),90,WorkflowCase_JMP);
					END_IF
				END_IF
			END_IF;

		(* Case 10 *)
		10:	
			(* Stato delle piazzole: valuto se sono tutte occupate in modo da segnalarlo all'operatore mediante lampeggio *)
			//////AllWABusy := TFCheckPalletFull(WorkArea:=WorkArea,WorkAreaState:=WorkAreaState,WorkPickPointState:=WorkPickPointState,Forming:=Forming); 
			(* Reset stati e missioni *)
			Mission^.State := MISSION_STATE_NOP;
			WorkAreaManager^.State := WAMANAGER_NOP;
			Ciclo_Di_Riposo.Stato			:= ANNULLATO;
			Ciclo_Prelievo_Lastra.Stato 	:= ANNULLATO;
			//Ciclo_Pelievo_Pallet.Stato 	:= ANNULLATO;
			Ciclo_Pelievo_Falda.Stato 		:= ANNULLATO;
			Ciclo_Deposito_Lastra.Stato 	:= ANNULLATO;
			//Ciclo_Deposito_Pallet.Stato 	:= ANNULLATO;
			Ciclo_Deposito_Falda.Stato 	:= ANNULLATO;
			ProductOnGripper 				:= KNOPRODUCT;
			TFWorkFlowCase(ADR(WorkFlow[0]),1,WorkflowCase_INC);

		(* Case 11 *)
		11:	TFWorkFlowCase(ADR(WorkFlow[0]),1,WorkflowCase_INC);
		
		(* Case 12 *)
		12:
			TFParametersArrayClear(ADR(ParametersArray));
			TFCommandSend(CmdHOME,ParametersArray,Modules^.AX_Z.Cmd);
			TFWorkFlowCase(ADR(WorkFlow[0]),1,WorkflowCase_INC);
			
		(* Case 13 *)	
		13:	IF TFStateCodeGet(Modules^.AX_Z.State) = StateHOME_END THEN
				TFParametersArrayClear(ADR(ParametersArray));
				ParametersArray.Parameters[0] := '100';
				ParametersArray.Parameters[1] := '13';
				Modules^.AX_Y.AxisPar^.Quota_Destinazione := WorkSpace^.Y/2 + OffSetPosYReposo;
				TFCommandSend(CmdMAN,ParametersArray,Modules^.AX_Y.Cmd);
				TFWorkFlowCase(ADR(WorkFlow[0]),1,WorkflowCase_INC);
			ELSIF CmdExe.RapidStopRequest > 0 OR TFPalletizerIsModuleError(Modules) THEN
				CmdExe.PhaseStopRequest := 1;
				CmdExe.RapidStopRequest := 1;
				TFWorkFlowCase(ADR(WorkFlow[0]),StateWF_ERROR,WorkflowCase_JMP);
			END_IF
			
		(* Case 14 *)
		14:
			IF TFStateCodeGet(Modules^.AX_Y.State) = StateMAN_END THEN
				TFCommandSend(CmdHOME,ParametersArray,Modules^.AX_X.Cmd);
				TFCommandSend(CmdHOME,ParametersArray,Modules^.AX_J.Cmd);
				TFCommandSend(CmdHOME,ParametersArray,Modules^.Pinza.Cmd);
				TFWorkFlowCase(ADR(WorkFlow[0]),20,WorkflowCase_JMP);
			ELSIF CmdExe.RapidStopRequest > 0 OR TFPalletizerIsModuleError(Modules) THEN
				CmdExe.PhaseStopRequest := 1;
				CmdExe.RapidStopRequest := 1;
				TFWorkFlowCase(ADR(WorkFlow[0]),StateWF_ERROR,WorkflowCase_JMP);
			END_IF
	
		(* Case 20 *)
		20:	IF TFStateCodeGet(Modules^.AX_X.State) = StateHOME_END AND
			TFStateCodeGet(Modules^.AX_J.State) = StateHOME_END AND 
			TFStateCodeGet(Modules^.Pinza.State) = StateHOME_END THEN
				TFCommandSend(CmdHOME,ParametersArray,Modules^.AX_Y.Cmd);
				TFWorkFlowCase(ADR(WorkFlow[0]),1,WorkflowCase_INC);
			ELSIF CmdExe.RapidStopRequest > 0 OR TFPalletizerIsModuleError(Modules) THEN
				CmdExe.PhaseStopRequest := 1;
				TFWorkFlowCase(ADR(WorkFlow[0]),StateWF_ERROR,WorkflowCase_JMP);
			END_IF
			
		(* Case 21 *)
		21:	IF TFStateCodeGet(Modules^.AX_Y.State) = StateHOME_END  THEN
				TFWorkFlowCase(ADR(WorkFlow[0]),1,WorkflowCase_INC);
			ELSIF CmdExe.RapidStopRequest > 0 OR TFPalletizerIsModuleError(Modules)  THEN
				CmdExe.PhaseStopRequest := 1;
				TFWorkFlowCase(ADR(WorkFlow[0]),StateWF_ERROR,WorkflowCase_JMP);
			END_IF
			
		(* Case 22 - *)
		22:	TFWorkFlowCase(ADR(WorkFlow[0]),90,WorkflowCase_JMP);
		
		(* Case 25 - Eseguo Home Direct *)
		25:
			TFParametersArrayClear(ADR(ParametersArray));
			ParametersArray.Parameters[0] := 'TRUE';//Il tipo di homing è HomeDirect
			TFPalletizerModulesCommandSend(CmdHOME,ParametersArray,Modules);
			TFWorkFlowCase(ADR(WorkFlow[0]),26,WorkflowCase_JMP);
			IF CmdExe.RapidStopRequest > 0 OR TFPalletizerIsModuleError(Modules)  THEN
				CmdExe.PhaseStopRequest := 1;
				CmdExe.RapidStopRequest := 1;
				TFWorkFlowCase(ADR(WorkFlow[0]),StateWF_ERROR,WorkflowCase_JMP);
			END_IF
		
		(* Case 26 - Attesa esecuzione HomeDirect *)
		26:	IF TFPalletizerModulesCheckState(StateHOME_END,Modules) THEN
				TFWorkFlowCase(ADR(WorkFlow[0]),90,WorkflowCase_JMP);
			ELSIF CmdExe.RapidStopRequest > 0 OR TFPalletizerIsModuleError(Modules)  THEN
				CmdExe.PhaseStopRequest := 1;
				TFWorkFlowCase(ADR(WorkFlow[0]),StateWF_ERROR,WorkflowCase_JMP);
			END_IF
			
		(* Case 90 - HomeDone *)
		90:	
			//Faccio partire tutti i WF dal case 0				
			FOR wfindx := 1 TO MAXWORKFLOW DO
				TFWorkFlowCase(ADR(WorkFlow[wfindx]),0,WorkflowCase_JMP);
			END_FOR
			
			IF NOT IN.PX_WorkArea[1] THEN
			// Pulisco piazzola in seguito ad estrazione
				TFClearWorkAreaArray(WorkArea,WorkAreaState,1);
			END_IF
			
			TFWorkFlowCase(ADR(WorkFlow[0]),94,WorkflowCase_JMP);
			
		(* Case 91 - Clear WorkArea *)
		
		91:	FOR k:= 1 TO MAXAREAPRESENT DO//(MAXAREA/2) DO
				IF NOT IN.PX_WorkArea[k] THEN
					// Pulisco piazzola in seguito ad estrazione
					TFClearWorkAreaArray(WorkArea,WorkAreaState,k);
				ELSE
					// preparo la piazzola solo se di tipo catasta pallet o layer	
					(*IF WorkArea^[k].Typology = TYPOLOGY_STACK OR WorkArea^[k].Typology = TYPOLOGY_LAYER  THEN
						//TFClearWorkAreaStack(WorkArea,WorkAreaState,k);
						IF (AutoToMan OR GateAcces) AND WorkArea^[k].Typology = TYPOLOGY_LAYER THEN
							WorkAreaState^[k].Learn_Z := ALTEZZA_CATASTA_FALDE;
							WorkAreaState^[k].Learned_Z := WorkAreaState^[k].Learn_Z;
							WorkAreaState^[k].H := ALTEZZA_CATASTA_FALDE;
							WorkAreaState^[k].DoLearn_Z := 1;	// Apprendimento da effettuare
						ELSIF ((AutoToMan OR GateAcces) AND WorkArea^[k].Typology = TYPOLOGY_STACK) OR (WorkAreaState^[k].H = 0 AND WorkArea^[k].Typology = TYPOLOGY_STACK) THEN	
							WorkAreaState^[k].Learn_Z := ALTEZZA_CATASTA_VUOTI;
							WorkAreaState^[k].Learned_Z := WorkAreaState^[k].Learn_Z;
							WorkAreaState^[k].H := ALTEZZA_CATASTA_VUOTI;
							WorkAreaState^[k].DoLearn_Z := 1;	// Apprendimento da effettuare						
						END_IF
					ELSIF WorkArea^[k].Typology = TYPOLOGY_PALLET AND Mission^.State = MISSION_STATE_NOP THEN
						IF WorkArea^[k].Enable <> 0 AND (WorkAreaState^[k].State = WORKAREA_STATE_FREE_DISABLED OR WorkAreaState^[k].State = WORKAREA_STATE_FREE_WORKING) THEN
							CmdExe.PhaseStopRequest := 1;
							WorkFlow[0].Enable := FALSE;
							TFError(ErrPALLETALREADYPRESENT,k,ADR(CmdExe),ADR(State),ADR(Error),ADR(ErrorLog));
						END_IF
					END_IF*)
				END_IF
			END_FOR
			TFWorkFlowCase(ADR(WorkFlow[0]),94,WorkflowCase_JMP);
			
			(* Case 94 - Clear WorkArea seconda metà *)
			94:
				PalletStackEmpty := 0;
				LayerStackEmpty := 0;
				GateAcces := FALSE;
				IF QuotaFuoriIngombro_X_AVUOTO = 0 THEN
					QuotaFuoriIngombro_X_AVUOTO := WorkPickPoint^[1].X;
				END_IF
				IF QuotaFuoriIngombro_Y_AVUOTO = 0 THEN
					QuotaFuoriIngombro_Y_AVUOTO := WorkPickPoint^[1].Y;
				END_IF
				IF QuotaFuoriIngombro_Z_AVUOTO = 0 THEN
					QuotaFuoriIngombro_Z_AVUOTO := WorkPickPoint^[1].Z + 300;
				END_IF
				//IF QuotaFuoriIngombro_J_AVUOTO = 0 THEN
				//	QuotaFuoriIngombro_J_AVUOTO := 90;
				//END_IF
				(* Inizializzo le quote di sicurezza ad un valore fittizzio elevato in modo da evitare possibili collisioni in caso di errore di calcolo.. NON dovrebbe mai accadere *)
				ErroreDiInterferenza := TFControlloInterferenza( Traiettoria := Traiettoria,
																WorkSpace := WorkSpace,
																WorkFootprint := WorkFootprint,
																WorkPickPoint := WorkPickPoint,
																WorkArea := WorkArea,
																Pallet := Pallet,
																Layer := Layer,
																Forming := Forming,
																Mission := Mission,
																WorkAreaManager := WorkAreaManager,
																ModuleAX_X := ADR(Modules^.AX_X),
																ModuleAX_Y := ADR(Modules^.AX_Y),
																ModuleAX_Z := ADR(Modules^.AX_Z),
																ModuleAX_J := ADR(Modules^.AX_J));
				
				//QuotaFuoriIngombro_Z_AVUOTO 	:= WorkSpace^.Z - 100;
				//QuotaFuoriIngombro_Z_ConFALDA 	:= WorkSpace^.Z - 100;
				//QuotaFuoriIngombro_Z_ConPEZZO 	:= WorkSpace^.Z - 100;
				//QuotaFuoriIngombro_Z_ConPALLET 	:= WorkSpace^.Z - 100;
				IF ErroreDiInterferenza > 0 THEN
				(* Se l'errore di interferenza è maggiore di 0, assegno alla traiettoria e alla missione dei i valori del punto di riposo, 
					in questo modo sbianco le eventuali quote non ammesse *)	
					CASE TIPOLOGIA_FUNZIONAMENTO_MACCHINA OF

						FUNZIONAMENTO_PALLETTIZZATORE:
							X_Riposo	:= WorkPickPoint^[1].X;
							Y_Riposo	:= WorkPickPoint^[1].Y + Dimensioni_Pinza.Larghezza;
							Z_Riposo	:= WorkPickPoint^[1].Z + OffsetSicurezza.Z.Avuoto;
							J_Riposo	:= 90;
						FUNZIONAMENTO_DEPAL:

							X_Riposo	:= WorkArea^[1].X;
							Y_Riposo	:= Workarea^[1].Y;
							Z_Riposo	:= 2000;                           
							J_Riposo	:= 90;                             

					
					END_CASE
			


					
					Traiettoria^.EndPoint.X := X_Riposo;
					Traiettoria^.EndPoint.Y := Y_Riposo;
					Traiettoria^.EndPoint.Z := Z_Riposo;
					Traiettoria^.EndPoint.J := J_Riposo;
					
					Mission^.PPick			:= PICKPOINT1;
					Mission^.TPick 			:= TPICK_NOT_DEFINED;
					Mission^.XPick 			:= X_Riposo;
					Mission^.YPick 			:= Y_Riposo;
					Mission^.ZPick 			:= Z_Riposo;
					Mission^.JPick 			:= J_Riposo;
					
					Mission^.XPlace := X_Riposo;
					Mission^.YPlace := Y_Riposo;
					Mission^.ZPlace := Z_Riposo;
					Mission^.JPlace := J_Riposo;
					ErroreDiInterferenza := 0;
				END_IF
				
				TFWorkFlowCase(ADR(WorkFlow[0]),100,WorkflowCase_JMP);
				
		(* Case 100 *)
		(* WorkFlow END *)
		100:WorkFlow[0].State := StateWF_END;
			WorkFlow[0].Enable := FALSE;
			OUT.HomeDone := TRUE;
			AutoToMan := FALSE;
			AssiInterpolati := FALSE;
			TFWorkFlowCase(ADR(WorkFlow[0]),0,WorkflowCase_JMP);

		(* Case 999 *)
		(* WorkFlow ERROR *)
		StateWF_ERROR:
			TFWorkFlowError(ADR(WorkFlow[0]),ADR(WorkFlowErrorLog[0]));
			WorkFlow[0].Enable := FALSE;

		ELSE
			TFWorkFlowError(ADR(WorkFlow[0]),ADR(WorkFlowErrorLog[0]));
			TFError(ErrNOCMDCASE,ErrNULL,ADR(CmdExe),ADR(State),ADR(Error),ADR(ErrorLog));

	END_CASE;
		
END_IF

(*-------------------------------------------------------------------------------------------*)		
(* WorkFlow 1 -  *)
(*-------------------------------------------------------------------------------------------*)
IF WorkFlow[1].Enable THEN

	IF NOT TFCommandCaseIsEnable(ADR(CmdExe)) THEN RETURN; END_IF
	CASE WorkFlow[1].WFCase OF

		(* Case 0 *)
		0: 	WorkFlow[1].State := StateWF_RUN;
			TFWorkFlowCase(ADR(WorkFlow[1]),1,WorkflowCase_INC);

		(* Case 1 *)
		1:	IF CmdExe.RapidStopRequest > 0 OR
				CmdExe.PhaseStopRequest > 0 THEN
				TFWorkFlowCase(ADR(WorkFlow[1]),100,WorkflowCase_JMP);
			ELSE
				(* Check Modules Error *)
				IF CmdExe.RapidStopRequest > 0 OR
					TFPalletizerIsModuleError(Modules) THEN
						TFParametersArrayClear(ADR (ParametersArray));
						TFPalletizerModulesCommandSend(CmdSTOP,ParametersArray,Modules);
						//CmdExe.PhaseStopRequest := 1;
						WorkFlow[1].Enable := FALSE;
				ELSE
					TFWorkFlowCase(ADR(WorkFlow[1]),9,WorkflowCase_JMP);	
				END_IF
			END_IF;
			
		(* Case 9 - Controllo che tutti i cicli siano ANNULLATI oppoure TERMINATI.. 
			Se sono INTERROTTI genero allarme affinchè in manuale, non aprono la pinza per annullare TUTTI i cicli!!*)	
		9:	 IF ((Ciclo_Prelievo_Lastra.Stato 	= ANNULLATO OR Ciclo_Prelievo_Lastra.Stato 	= TERMINATO) AND
				(Ciclo_Pelievo_Falda.Stato 		= ANNULLATO OR Ciclo_Pelievo_Falda.Stato	= TERMINATO) AND
				(Ciclo_Deposito_Lastra.Stato	= ANNULLATO OR Ciclo_Deposito_Lastra.Stato 	= TERMINATO) AND
				(Ciclo_Deposito_Falda.Stato		= ANNULLATO OR Ciclo_Deposito_Falda.Stato 	= TERMINATO) AND 
				(Ciclo_Di_Riposo.Stato			= ANNULLATO OR Ciclo_Di_Riposo.Stato 		= TERMINATO) AND
				(Ciclo_Prelievo_Lastra_Depal.Stato = ANNULLATO OR Ciclo_Prelievo_Lastra_Depal.Stato = TERMINATO) AND
				(Ciclo_Deposito_Lastra_Depal.Stato = ANNULLATO OR Ciclo_Deposito_Lastra_Depal.Stato = TERMINATO OR (Ciclo_Deposito_Lastra_Depal.Passo = 56 AND Ciclo_Deposito_Lastra_Depal.Stato = INTERROTTO)) AND
				(Ciclo_Deposito_Falda_Depal.Stato = ANNULLATO OR Ciclo_Deposito_Falda_Depal.Stato = TERMINATO)) THEN
				WaitPositionRequest := FALSE;
				IF Mission^.State = MISSION_STATE_NOP THEN
					MissionStateCase^.NCase := 0;
					MissionStateCase^.Mission := MISSION_STATE_NOP;
				END_IF
				TFWorkFlowCase(ADR(WorkFlow[1]),1,WorkflowCase_INC);
			ELSE
				TFError(ErroreMANCATO_RESET_MISSIONI,ErrNULL,ADR(CmdExe),ADR(State),ADR(Error),ADR(ErrorLog));
				CmdExe.RapidStopRequest := 1;
				WorkFlow[1].Enable := FALSE;
			END_IF
				
		(* Case 10 *)	
		10:	(* Check Modules Error *)
			IF CmdExe.RapidStopRequest > 0 OR
				TFPalletizerIsModuleError(Modules) THEN
					WorkFlow[1].Enable := FALSE;
			ELSIF (CmdExe.PhaseStopRequest > 0 AND 
					((Mission^.State = MISSION_STATE_NOP AND (InWaitPosition OR (Ciclo_Deposito_Lastra_Depal.Passo = 56 AND Ciclo_Deposito_Lastra_Depal.Stato = INTERROTTO))) OR
						(Mission^.State = MISSION_STATE_DEPOSITO_LASTRA_DEPAL_RUN AND (Ciclo_Deposito_Lastra_Depal.Passo = 56 AND Ciclo_Deposito_Lastra_Depal.Stato = INTERROTTO)))) THEN
					CmdExe.PhaseStopRequest :=1;
					TFWorkFlowCase(ADR(WorkFlow[1]),100,WorkflowCase_JMP);	
			ELSE
				TFTimerCall(ADR(TimerPacchi1Minuto),Cfg.TimeBase);
				TFTimerSet(ADR(TimerPacchi1Minuto),60000,NOT AttivaTimerContaPacchi1Minuto);
				TFTimerCall(ADR(TimerPacchi5Minuti),Cfg.TimeBase);
				TFTimerSet(ADR(TimerPacchi5Minuti),300000,NOT AttivaTimerContaPacchi5Minuti);
				IF TFTimerDone(ADR(TimerPacchi1Minuto)) THEN
					TimerDone1 := TimerDone1 +1;
					AttivaTimerContaPacchi1Minuto := FALSE;
					PacchiPrelevatiAlMinuto := Pacchi1Minuto;
					PacchiAlMinuto[TimerDone1] := PacchiPrelevatiAlMinuto;	
					Pacchi1Minuto := 0;					
				END_IF
				IF TFTimerDone(ADR(TimerPacchi5Minuti)) THEN
					AttivaTimerContaPacchi5Minuti := FALSE;
					PacchiPrelevatiIn5MinutiAppoggio := 0;
					FOR cuontpac := 1 TO TimerDone1 DO
						PacchiPrelevatiIn5MinutiAppoggio := PacchiPrelevatiIn5MinutiAppoggio + PacchiAlMinuto[cuontpac];
						PacchiAlMinuto[cuontpac] := 0;
					END_FOR	
					IF TimerDone1 > 0 AND PacchiPrelevatiIn5MinutiAppoggio > 0 THEN
						PacchiPrelevatiIn5Minuti := PacchiPrelevatiIn5MinutiAppoggio / TimerDone1;
						TimerDone1 := 0;
					END_IF		
				END_IF
				(* Filtro fotocellula presenza materiale su pinza *)
				(*Filtro_PX_GripPresence(IN_Signal := PX_GripPresence,
										FilterTime_ON := 400,
										FilterTime_OFF := 500,
										OUT_Signal_Filtrato => PX_GripPresenceFiltrata);
				//*)
				//PX_GripPresenceFiltrata := PX_GripPresence;
				PX_GripPresenceFiltrata := Modules^.Pinza.StatoPinza.ElementoPrelevato;
				(* Stato delle piazzole: valuto se sono tutte occupate in modo da segnalarlo all'operatore mediante lampeggio *)
				//AllWABusy := TFCheckPalletFull(WorkArea,WorkAreaState,WorkPickPointState); 
				
				(* Controllo se nella postazione pallet e falde è presente il materiale *)	
				PalletStackEmpty := 0;// TFCheckPalletPresence(WorkArea,WorkAreaState,IN.PX_WorkArea);
				LayerStackEmpty := 0;//NOT IN.PX_WorkArea[NumPostazioneFALDE];  TFCheckLayerPresence(WorkArea,WorkAreaState,IN.PX_WorkArea);
				//IF LayerStackEmpty > 0 OR (IN.PX_WorkArea[NumPostazioneFALDE] AND WorkAreaManager^.State = WAMANAGER_NOP)THEN
				//	CmdExe.RapidStopRequest := 1;
				//	TFError(ErrMODULEPALLETIZERROBOT_EMPTYLAYERSTACK,PalletLayerPresence,ADR(CmdExe),ADR(State),ADR(Error),ADR(ErrorLog));
				//END_IF
				
				(* Set della richiesta della posizione di  riposo da inviare al WAM *)		
				WaitPositionRequest := (WaitPositionRequest OR ExternalWaitPositionRequest OR CmdExe.PhaseStopRequest > 0);
				

				
				TFCalcoliFuoriIngombri.StatoWAM_precedente := WorkAreaManager^.State;//Setto lo stato del wam prima che venga elaborato il FB
				
				(* Chiamata del FB che gestisce il Pallettizzatore osservendo lo stato delle varie Work Area e del Pallettizatore stesso *)		
				TFPalletizerWorkAreaManagerTF(	Cfg 			:= Cfg,
												WorkArea 		:= WorkArea,
												WorkAreaState 	:= WorkAreaState,
												WorkAreaOffset	:= WorkAreaOffset,
												PX_WorkArea 	:= IN.PX_WorkArea,
												WorkPickPoint 	:= WorkPickPoint,
												WorkPickPointState := WorkPickPointState,
												WorkAreaProductionList := WorkAreaProductionList,
												//WorkPickPointStoreState:= WorkPickPointStoreState,
												//WorkPickPointTransportState := WorkPickPointTransportState,
												WorkPickPointOffset := WorkPickPointOffset,
												Forming 		:= Forming,
												Pallet 			:= Pallet,
												Layer 			:= Layer,
												Mission 		:= Mission,
												PickPlaceParameters 		:= PickPlaceParameters,
												ExternalWaitPositionRequest := WaitPositionRequest,
												ProgressiveNrWA 		:= ProgressiveNrWA,
												UsedCode				:= UsedCode,
												TCPParameter 			:= TCPParameter,
												TilterPack 				:= TilterPack,
												PreviousPWA 			:= PreviousPWA,
												RestoreCWA 				:= RestoreCWA,
												PreviousStackWA 		:= PreviousStackWA,
												WorkAreaManager 		:= WorkAreaManager,
												ModuleAX_X 				:= ADR(Modules^.AX_X),
												ModuleAX_Y 				:= ADR(Modules^.AX_Y),
												ModuleAX_Z 				:= ADR(Modules^.AX_Z),
												ModuleAX_J 				:= ADR(Modules^.AX_J),
												ModulePinza           	:= ADR(Modules^.Pinza),
												WorkAreaZone			:= WorkAreaZone,
												GestioneAZoneAbilitata 	:= GestioneAZoneAbilitata, 
												//HandlingPackTable 		:= HandlingPackTable,
												ArrayPacchi				:= ArrayPacchi,
												HandlingRun				:= IN.HandlingRun,
												//RichiestaStartRibaltino := RichiestaStartRibaltino,
												AbilitaForzaturaStatoDaRiposoAPrelievo 			:= AbilitaForzaturaStatoWAMDaCicloRiposoACicloPrelievo,
												AbilitaDisposizionePalletContinua 				:= AbilitaDisposizionePalletContinua,
												AbilitaDepositoPaccoOrrizzonataleConTasteggio 	:= AbilitaDepositoPaccoOrrizzonataleConTasteggio,
												AbilitaOffsetInUscitaTasteggioPrelievoPallet 	:= AbilitaOffsetInUscitaTasteggioPrelievoPallet,
												RichiestaIngZonaDX 								:= RichiestaIngZonaDX, 
												RichiestaIngZonaSX 								:= RichiestaIngZonaSX,
												InWaitPosition									=> InWaitPosition,
												DepositoPaccoInLenta							=> DepositoPaccoInLenta,
												ForzaPrelievoPaccoDuranteCicloDiRiposo 			=> ForzaPrelievoPaccoDuranteCicloDiRiposo,);

				(* Valuto se il WAMANAGER ha un errore, in tal caso blocco tutto *)								
				IF TFPalletizerWorkAreaManagerTF.Errore.Code > 0 THEN
					CmdExe.PhaseStopRequest := 1;
					WorkFlow[1].Enable := FALSE;
					TFError(TFPalletizerWorkAreaManagerTF.Errore.Code,TFPalletizerWorkAreaManagerTF.Errore.ExtraCode,ADR(CmdExe),ADR(State),ADR(Error),ADR(ErrorLog));
				END_IF

				(* Chiamata della Function che assegna le volocità ai vari assi *)	
				IF (NOT AssiInterpolati	AND AbilitaInterpolazioneAssi^) OR NOT AbilitaInterpolazioneAssi^ THEN					
					TFCalcoloVelocita(AxisOverride := AxisOverride, 
													Mission := Mission,
													ArrayPacchi		 := ArrayPacchi,
													DepositoPaccoInLenta := DepositoPaccoInLenta);
				END_IF
				
				//#################################################################################################
				//#################################################################################################
				(* Chiamata della FB che definisce le quote necessarie a compiere la traiettoria della missione in corso *)
				TFCalcoloTraiettoria(	Traiettoria := Traiettoria,
										WorkSpace := WorkSpace,
										WorkFootprint := WorkFootprint,
										WorkPickPoint := WorkPickPoint,
										WorkAreaState := WorkAreaState,
										WorkPickPoint := WorkPickPoint,
										WorkPickPointState := WorkPickPointState,
										WorkPickPointDimension := WorkPickPointDimension,
										WorkArea := WorkArea,
										Pallet := Pallet,
										Layer := Layer,
										Forming := Forming,
										Mission := Mission,
										WorkAreaManager := WorkAreaManager,
										ModuleAX_X := ADR(Modules^.AX_X),
										ModuleAX_Y := ADR(Modules^.AX_Y),
										ModuleAX_Z := ADR(Modules^.AX_Z),
										ModuleAX_J := ADR(Modules^.AX_J));
				(* Calcolo dell'ingombro delle colonne centrali*)						
				TFCalcoliFuoriIngombri(  Traiettoria := Traiettoria,
										WorkSpace := WorkSpace,
										WorkFootprint := WorkFootprint,
										WorkPickPoint := WorkPickPoint,
										//WorkPickPointState := WorkPickPointState,
										WorkPickPointDimension := WorkPickPointDimension,
										WorkArea := WorkArea,
										WorkAreaState := WorkAreaState,
										WorkAreaOffset:= WorkAreaOffset,
										Pallet := Pallet,
										Layer := Layer,
										Forming := Forming,
										PickPlaceParameters:=PickPlaceParameters,
										Mission := Mission,
										WorkAreaManager := WorkAreaManager,
										ModuleAX_X := ADR(Modules^.AX_X),
										ModuleAX_Y := ADR(Modules^.AX_Y),
										ModuleAX_Z := ADR(Modules^.AX_Z),
										ModuleAX_J := ADR(Modules^.AX_J),
										PX_WorkArea 	:= IN.PX_WorkArea,
										AbilitaCalcoloIngombroOttimizzato := AbilitaCalcoloIngombroOttimizzato^);						
					



				(* Reset delle momorie di quota raggiunta(per sicurezza..)*)						
				QuotaAnticipoDinamicaX_Raggiunta := FALSE; 
				QuotaAnticipoDinamicaY_Raggiunta := FALSE; 
				QuotaAnticipoDinamicaZ_Raggiunta := FALSE; 
				QuotaAnticipoDinamicaJ_Raggiunta := FALSE;
				(* Calcolo delle quote di anticipo *)
				(*TFCalcoloPuntiDiAnticipoDinamici(	Traiettoria := Traiettoria,
													WorkSpace := WorkSpace,
													WorkFootprint := WorkFootprint,
													WorkPickPoint := WorkPickPoint,
													WorkPickPointState := WorkPickPointState,
													WorkPickPointOffset := WorkPickPointOffset,
													WorkPickPointDimension := WorkPickPointDimension,
													WorkArea := WorkArea,
													WorkAreaState := WorkAreaState,
													Pallet := Pallet,
													Layer := Layer,
													Forming := Forming,
													PickPlaceParameters:=PickPlaceParameters,
													Mission := Mission,
													WorkAreaManager := WorkAreaManager,
													ModuleAX_X := ADR(Modules^.AX_X),
													ModuleAX_Y := ADR(Modules^.AX_Y),
													ModuleAX_Z := ADR(Modules^.AX_Z),
													ModuleAX_J := ADR(Modules^.AX_J),
													AbilitaAnticipoDinamico := AbilitaAnticipoDinamico^);*)
												
				(* Valutazione se gli assi sono in finestra di PassMode *) 
				TFValutaAssiInFinestraDiPassMode(	ModuleAX_X := ADR(Modules^.AX_X),
													ModuleAX_Y := ADR(Modules^.AX_Y),
													ModuleAX_Z := ADR(Modules^.AX_Z),
													ModuleAX_J := ADR(Modules^.AX_J),
													WorkAreaManager := WorkAreaManager,
													Traiettoria := Traiettoria);
									
				(* Chiamata della function che controlla che i valori assunti dalle quote non vadano fuori dai limiti e non vi sia collisione tra pinza e oggetti *)						
				
				IF WorkAreaManager^.State <> WAMANAGER_NOP AND WorkAreaManager^.State <> WAMANAGER_CICLO_RIPOSO_INIT AND WorkAreaManager^.State <> WAMANAGER_CICLO_LASTRA_PP_INIT THEN
					ErroreDiInterferenza := TFControlloInterferenza( Traiettoria := Traiettoria,
											WorkSpace := WorkSpace,
											WorkFootprint := WorkFootprint,
											WorkPickPoint := WorkPickPoint,
											WorkArea := WorkArea,
											Pallet := Pallet,
											Layer := Layer,
											Forming := Forming,
											Mission := Mission,
											WorkAreaManager := WorkAreaManager,
											ModuleAX_X := ADR(Modules^.AX_X),
											ModuleAX_Y := ADR(Modules^.AX_Y),
											ModuleAX_Z := ADR(Modules^.AX_Z),
											ModuleAX_J := ADR(Modules^.AX_J));	
				END_IF
				(* Controllo che non sia settata la memoria di Errore Di Interferenza *)							
				IF ErroreDiInterferenza > 0 THEN
					TFError(ErroreDiInterferenza,ErrNULL,ADR(CmdExe),ADR(State),ADR(Error),ADR(ErrorLog));
					CmdExe.RapidStopRequest := 1;
				ELSIF TFCalcoliFuoriIngombri.Errore > 0 THEN
					TFError(TFCalcoliFuoriIngombri.Errore,ErrNULL,ADR(CmdExe),ADR(State),ADR(Error),ADR(ErrorLog));
					CmdExe.RapidStopRequest := 1;
				END_IF
								
				(* Verifico se la pinza se è in quota di fuori-Ingombro e setto un bit *)
				PinzaInQuotaFuoriIngombro := TFFuoriIngombroVerticaleOK(Modules^.AX_Z.Ax^.AxRef^.NcToPlc.SetPos,Mission);
				(* Se la quota dell'asse Z è inferiore alla quaota di deposito + 100 mm, disabilito il controllo.
					In questo modo non ho falsi errori in fase di deposito *)
				AbilitaControlloPHGripPresence := AbilitaControlloPHGripPresence AND PinzaInQuotaFuoriIngombro;//Modules^.AX_Z.Ax^.AxRef^.NcToPlc.SetPos >= Mission^.ZPlace + 100;	
	
				PinzaConProdottoInPresa := Modules^.Pinza.StatoPinza.LatoDxPiastrellaInPresa AND Modules^.Pinza.StatoPinza.LatoSxPiastrellaInPresa OR ProductOnGripper <> KNOPRODUCT;

				(* Set Stato Missione in base allo stato del Work Area Manager*)
				CASE WorkAreaManager^.State OF					
					WAMANAGER_NOP:
						//WorkPickPointState^[Mission^.PPick].TC := 0;
						//DepositoFaldaSuCatastaVuoti := FALSE;
						Mission^.State := MISSION_STATE_NOP;
						MissionStateCase^.NCase := 0;
						MissionStateCase^.Mission := MISSION_STATE_NOP;

						//ResetComandoRibaltinoEseguito := FALSE;
						
						(* Verifica che vi siano falda e pallet con codice uguali a quello delle foratura attiva *)
						//PalletLayerPresence := TFPalletizerCheckPalletLayerCode(WorkArea,WorkAreaState,Forming);
						//IF PalletLayerPresence > 0 THEN
						//	CmdExe.PhaseStopRequest := 1;
						//	WorkFlow[1].Enable := FALSE;
						//	TFError(PalletLayerPresence,ErrNULL,ADR(CmdExe),ADR(State),ADR(Error),ADR(ErrorLog));
						//END_IF
						
						IF Modules^.AX_Z.Ax^.Status.ActPosition >= QuotaFuoriIngombro_Z_AVUOTO - 5 OR Modules^.AX_Z.Ax^.Status.ActPosition >= QuotaFuoriIngombro_Z_ConPEZZO - 5 THEN
							PinzaInQuotaFuoriIngombroPerTrasporti := TRUE;
						//ELSE
						//	PinzaInQuotaFuoriIngombroPerTrasporti := FALSE;
						END_IF
					{Region "WA MANAGER RIPOSO"}													
					WAMANAGER_CICLO_RIPOSO_RUN:
						(* Controllo che la pinza si libera *)
						IF AbilitaControlloPHGripPresence THEN
							IF PinzaConProdottoInPresa THEN
								CmdExe.RapidStopRequest := 1;
								TFError(ErrPRESENZA_MATERIALE_SUPINZA_CICLO_RIPOSO,ErrNull,ADR(CmdExe),ADR(State),ADR(Error),ADR(ErrorLog));
							ELSE
								Mission^.State := MISSION_STATE_VAIaRIPOSO_RUN;
							END_IF
						ELSE
							PX_GripPresenceOK := TRUE;
							Mission^.State := MISSION_STATE_VAIaRIPOSO_RUN;
						END_IF
						(* Quando Sono Fuori ingombro setto il FI x il ribaltino *)
						IF (Modules^.AX_Z.Ax^.Status.ActPosition >= QuotaFuoriIngombro_Z_AVUOTO - 5 OR Modules^.AX_Z.Ax^.Status.ActPosition >= QuotaFuoriIngombro_Z_ConPEZZO - 5) AND
							 NOT ResetComandoRibaltinoEseguito THEN
								PinzaInQuotaFuoriIngombroPerTrasporti := TRUE;
								ResetComandoRibaltinoEseguito := TRUE;
						END_IF
																				
					WAMANAGER_CICLO_RIPOSO_END:
						PX_GripPresenceOK := FALSE;
						Mission^.State := MISSION_STATE_NOP;
						ProductOnGripper := KNOPRODUCT;
					{endregion}
					{Region "WA MANAGER FALDA"}
					WAMANAGER_CICLO_PRELIEVO_FALDA_RUN:
						OUT.StartTilter := FALSE;
						//DepositoFaldaSuCatastaVuoti := TRUE;
						Modules^.AX_Z.AbilitaOffsetInUscitaTasteggio := FALSE;
						
						IF AbilitaControlloPHGripPresence THEN
							IF (PX_GripPresenceFiltrata AND NOT PX_GripPresenceOK) AND PinzaInQuotaFuoriIngombro THEN
								TFError(ErrPRESENZA_MATERIALE_SUPINZA_CICLO_PRELFALDA,ErrPRESENZA_MATERIALE_SUPINZA_CICLO_PRELFALDA,ADR(CmdExe),ADR(State),ADR(Error),ADR(ErrorLog));
								CmdExe.RapidStopRequest := 1;
							ELSE
								PX_GripPresenceOK := TRUE;
								Mission^.State := MISSION_STATE_PRELIEVO_FALDA_RUN;
							END_IF
						ELSE
							PX_GripPresenceOK := TRUE;
							Mission^.State := MISSION_STATE_PRELIEVO_FALDA_RUN;
						END_IF
												
					WAMANAGER_CICLO_PRELIEVO_FALDA_END:
						OUT.StartTilter := FALSE;
						PX_GripPresenceOK := FALSE;
						//DepositoFaldaSuCatastaVuoti := FALSE;
						Mission^.State := MISSION_STATE_DEPOSITO_FALDA_RUN;
						ProductOnGripper := KPRODUCTLOADED;
				   							
					WAMANAGER_CICLO_DEPOSITO_FALDA_RUN:
						OUT.StartTilter := FALSE;
						//DepositoFaldaSuCatastaVuoti := FALSE;
						Modules^.AX_Z.AbilitaOffsetInUscitaTasteggio := FALSE;
						
						(* Se è abilitato il controllo della presenza utilizzando la fotocellula *)
						IF AbilitaControlloPHGripPresence THEN
							(* Se NON vedo la fotocellula e ho memorizzato di avere un prodotto *)
							IF not PX_GripPresenceFiltrata AND ProductOnGripper = KPRODUCTLOADED THEN
								TFError(ErrLOADLOST,ErrNULL,ADR(CmdExe),ADR(State),ADR(Error),ADR(ErrorLog));
								CmdExe.RapidStopRequest := 1;
							END_IF
						END_IF	
						
						(* Se non ho rilevato alcun errore procedo con la missione *)
						IF CmdExe.RapidStopRequest <> 1 THEN
								Mission^.State := MISSION_STATE_DEPOSITO_FALDA_RUN;
						END_IF
					
					WAMANAGER_CICLO_DEPOSITO_FALDA_END:
						OUT.StartTilter := FALSE;
						ProductOnGripper := KNOPRODUCT;
					{endregion}		

